LIN {X 0,Y 142.347,Z 443.787,A -85,B 0,C 180,E1 -25610.985,E2 -25610.985} C_VEL
LIN {X 0,Y 135.867,Z 450.599,A -85,B 0,C 180,E1 -25615.317,E2 -25615.317} C_VEL
LIN {X 0,Y 131.216,Z 455.128,A -85,B 0,C 180,E1 -25619.411,E2 -25619.411} C_VEL
LIN {X 0,Y 127.135,Z 458.6,A -85,B 0,C 180,E1 -25623.749,E2 -25623.749} C_VEL
LIN {X 0,Y 122.957,Z 461.7,A -85,B 0,C 180,E1 -25629.939,E2 -25629.939} C_VEL
LIN {X 0,Y 120.458,Z 463.257,A -85,B 0,C 180,E1 -25636.499,E2 -25636.499} C_VEL
LIN {X 0,Y 119.459,Z 463.204,A -85,B 0,C 180,E1 -25643.237,E2 -25643.237} C_VEL
LIN {X 0,Y 119.528,Z 462.151,A -85,B 0,C 180,E1 -25648.311,E2 -25648.311} C_VEL
LIN {X 0,Y 119.517,Z 460.979,A -85,B 0,C 180,E1 -25651.51,E2 -25651.51} C_VEL
LIN {X 0,Y 119.554,Z 458.203,A -85,B 0,C 180,E1 -25656.745,E2 -25656.745} C_VEL
LIN {X 0,Y 120.052,Z 454.435,A -85,B 0,C 180,E1 -25661.816,E2 -25661.816} C_VEL
LIN {X 0,Y 121.344,Z 449.309,A -85,B 0,C 180,E1 -25667.013,E2 -25667.013} C_VEL
LIN {X 0,Y 123.514,Z 443.317,A -85,B 0,C 180,E1 -25671.698,E2 -25671.698} C_VEL
LIN {X 0,Y 126.362,Z 435.566,A -85,B 0,C 180,E1 -25676.41,E2 -25676.41} C_VEL
LIN {X 0,Y 127.73,Z 431.92,A -85,B 0,C 180,E1 -25678.233,E2 -25678.233} C_VEL
LIN {X 0,Y 128.781,Z 427.935,A -85,B 0,C 180,E1 -25680.111,E2 -25680.111} C_VEL
LIN {X 0,Y 128.861,Z 421.063,A -85,B 0,C 180,E1 -25683.301,E2 -25683.301} C_VEL
LIN {X 0,Y 128.961,Z 413.731,A -85,B 0,C 180,E1 -25686.286,E2 -25686.286} C_VEL
LIN {X 0,Y 129.981,Z 408.956,A -85,B 0,C 180,E1 -25687.771,E2 -25687.771} C_VEL
LIN {X 0,Y 133.424,Z 398.451,A -85,B 0,C 180,E1 -25690.173,E2 -25690.173} C_VEL
LIN {X 0,Y 136.671,Z 386.681,A -85,B 0,C 180,E1 -25692.187,E2 -25692.187} C_VEL
LIN {X 0,Y 139.335,Z 373.81,A -85,B 0,C 180,E1 -25693.773,E2 -25693.773} C_VEL
LIN {X 0,Y 141.317,Z 360.485,A -85,B 0,C 180,E1 -25694.819,E2 -25694.819} C_VEL
LIN {X 0,Y 143.543,Z 329.086,A -85,B 0,C 180,E1 -25696.247,E2 -25696.247} C_VEL
LIN {X 0,Y 143.992,Z 319.506,A -85,B 0,C 180,E1 -25696.718,E2 -25696.718} C_VEL
LIN {X 0,Y 143.262,Z 306.343,A -85,B 0,C 180,E1 -25697.853,E2 -25697.853} C_VEL
LIN {X 0,Y 138.673,Z 293.214,A -85,B 0,C 180,E1 -25700.561,E2 -25700.561} C_VEL
LIN {X 0,Y 133.405,Z 281.529,A -85,B 0,C 180,E1 -25703.8,E2 -25703.8} C_VEL
LIN {X 0,Y 128.28,Z 273.681,A -85,B 0,C 180,E1 -25707.131,E2 -25707.131} C_VEL
LIN {X 0,Y 125.597,Z 269.89,A -85,B 0,C 180,E1 -25709.063,E2 -25709.063} C_VEL
LIN {X 0,Y 123.046,Z 266.259,A -85,B 0,C 180,E1 -25711.072,E2 -25711.072} C_VEL
LIN {X 0,Y 119.947,Z 262.642,A -85,B 0,C 180,E1 -25713.698,E2 -25713.698} C_VEL
LIN {X 0,Y 119.012,Z 260.746,A -85,B 0,C 180,E1 -25714.651,E2 -25714.651} C_VEL
LIN {X 0,Y 116.625,Z 258.914,A -85,B 0,C 180,E1 -25716.905,E2 -25716.905} C_VEL
LIN {X 0,Y 115.229,Z 256.404,A -85,B 0,C 180,E1 -25718.534,E2 -25718.534} C_VEL
LIN {X 0,Y 114.966,Z 255.164,A -85,B 0,C 180,E1 -25719.07,E2 -25719.07} C_VEL
LIN {X 0,Y 115.102,Z 255.137,A -85,B 0,C 180,E1 -25725.864,E2 -25725.864} C_VEL
LIN {X 0,Y 115.285,Z 255.125,A -85,B 0,C 180,E1 -25729.462,E2 -25729.462} C_VEL
LIN {X 0,Y 115.488,Z 255.097,A -85,B 0,C 180,E1 -25736.511,E2 -25736.511} C_VEL
LIN {X 0,Y 115.95,Z 254.997,A -85,B 0,C 180,E1 -25740,E2 -25740} C_VEL
LIN {X 0,Y 115.327,Z 255.113,A -85,B 0,C 180,E1 -25747.001,E2 -25747.001} C_VEL
LIN {X 0,Y 115.178,Z 255.094,A -85,B 0,C 180,E1 -25752.556,E2 -25752.556} C_VEL
LIN {X 0,Y 114.938,Z 255.142,A -85,B 0,C 180,E1 -25757.802,E2 -25757.802} C_VEL
LIN {X 0,Y 114.891,Z 255.162,A -85,B 0,C 180,E1 -25763.457,E2 -25763.457} C_VEL
LIN {X 0,Y 114.843,Z 255.178,A -85,B 0,C 180,E1 -25771.068,E2 -25771.068} C_VEL
LIN {X 0,Y 114.795,Z 255.21,A -85,B 0,C 180,E1 -25772.593,E2 -25772.593} C_VEL
LIN {X 0,Y 115.589,Z 257.654,A -85,B 0,C 180,E1 -25773.699,E2 -25773.699} C_VEL
LIN {X 0,Y 117.753,Z 260.059,A -85,B 0,C 180,E1 -25775.949,E2 -25775.949} C_VEL
LIN {X 0,Y 119.112,Z 260.981,A -85,B 0,C 180,E1 -25777.182,E2 -25777.182} C_VEL
LIN {X 0,Y 121.041,Z 264.197,A -85,B 0,C 180,E1 -25779.023,E2 -25779.023} C_VEL
LIN {X 0,Y 123.115,Z 266.362,A -85,B 0,C 180,E1 -25780.713,E2 -25780.713} C_VEL
LIN {X 0,Y 125.486,Z 269.811,A -85,B 0,C 180,E1 -25782.589,E2 -25782.589} C_VEL
LIN {X 0,Y 126.743,Z 271.497,A -85,B 0,C 180,E1 -25783.51,E2 -25783.51} C_VEL
LIN {X 0,Y 131.911,Z 279.095,A -85,B 0,C 180,E1 -25786.994,E2 -25786.994} C_VEL
LIN {X 0,Y 137.593,Z 288.613,A -85,B 0,C 180,E1 -25790.375,E2 -25790.375} C_VEL
LIN {X 0,Y 142.188,Z 297.608,A -85,B 0,C 180,E1 -25792.876,E2 -25792.876} C_VEL
LIN {X 0,Y 144.941,Z 303.696,A -85,B 0,C 180,E1 -25794.304,E2 -25794.304} C_VEL
LIN {X 0,Y 141.754,Z 350.025,A -85,B 0,C 180,E1 -25796.354,E2 -25796.354} C_VEL
LIN {X 0,Y 139.926,Z 363.432,A -85,B 0,C 180,E1 -25797.438,E2 -25797.438} C_VEL
LIN {X 0,Y 137.503,Z 376.255,A -85,B 0,C 180,E1 -25799.058,E2 -25799.058} C_VEL
LIN {X 0,Y 134.688,Z 387.934,A -85,B 0,C 180,E1 -25801.15,E2 -25801.15} C_VEL
LIN {X 0,Y 131.103,Z 399.265,A -85,B 0,C 180,E1 -25803.761,E2 -25803.761} C_VEL
LIN {X 0,Y 127.423,Z 409.472,A -85,B 0,C 180,E1 -25806.869,E2 -25806.869} C_VEL
LIN {X 0,Y 124.118,Z 417.825,A -85,B 0,C 180,E1 -25810.147,E2 -25810.147} C_VEL
LIN {X 0,Y 120.414,Z 426.872,A -85,B 0,C 180,E1 -25814.781,E2 -25814.781} C_VEL
LIN {X 0,Y 117.233,Z 434.194,A -85,B 0,C 180,E1 -25819.647,E2 -25819.647} C_VEL
LIN {X 0,Y 115.036,Z 440.041,A -85,B 0,C 180,E1 -25824.749,E2 -25824.749} C_VEL
LIN {X 0,Y 113.521,Z 444.662,A -85,B 0,C 180,E1 -25830.007,E2 -25830.007} C_VEL
LIN {X 0,Y 112.764,Z 447.542,A -85,B 0,C 180,E1 -25834.285,E2 -25834.285} C_VEL
LIN {X 0,Y 112.166,Z 450.75,A -85,B 0,C 180,E1 -25840.84,E2 -25840.84} C_VEL
LIN {X 0,Y 112.34,Z 451.922,A -85,B 0,C 180,E1 -25844.497,E2 -25844.497} C_VEL
LIN {X 0,Y 112.924,Z 452.662,A -85,B 0,C 180,E1 -25848.136,E2 -25848.136} C_VEL
LIN {X 0,Y 113.99,Z 453.051,A -85,B 0,C 180,E1 -25852.357,E2 -25852.357} C_VEL
LIN {X 0,Y 116.639,Z 452.5,A -85,B 0,C 180,E1 -25858.823,E2 -25858.823} C_VEL
LIN {X 0,Y 118.635,Z 451.603,A -85,B 0,C 180,E1 -25862.223,E2 -25862.223} C_VEL
LIN {X 0,Y 121.126,Z 450.227,A -85,B 0,C 180,E1 -25865.676,E2 -25865.676} C_VEL
LIN {X 0,Y 125.185,Z 447.493,A -85,B 0,C 180,E1 -25870.216,E2 -25870.216} C_VEL
LIN {X 0,Y 130.145,Z 443.612,A -85,B 0,C 180,E1 -25874.592,E2 -25874.592} C_VEL
LIN {X 0,Y 136.739,Z 437.557,A -85,B 0,C 180,E1 -25879.3,E2 -25879.3} C_VEL
LIN {X 0,Y 143.074,Z 430.847,A -85,B 0,C 180,E1 -25882.962,E2 -25882.962} C_VEL
LIN {X 0,Y 148.716,Z 423.972,A -85,B 0,C 180,E1 -25885.791,E2 -25885.791} C_VEL
LIN {X 0,Y 154.702,Z 415.627,A -85,B 0,C 180,E1 -25888.408,E2 -25888.408} C_VEL
LIN {X 0,Y 160.312,Z 406.479,A -85,B 0,C 180,E1 -25890.611,E2 -25890.611} C_VEL
LIN {X 0,Y 166.148,Z 395.072,A -85,B 0,C 180,E1 -25892.658,E2 -25892.658} C_VEL
LIN {X 0,Y 170.694,Z 383.759,A -85,B 0,C 180,E1 -25894.244,E2 -25894.244} C_VEL
LIN {X 0,Y 174.645,Z 371.716,A -85,B 0,C 180,E1 -25895.405,E2 -25895.405} C_VEL
LIN {X 0,Y 177.667,Z 358.526,A -85,B 0,C 180,E1 -25896.32,E2 -25896.32} C_VEL
LIN {X 0,Y 179.589,Z 345.087,A -85,B 0,C 180,E1 -25896.904,E2 -25896.904} C_VEL
LIN {X 0,Y 180.483,Z 334.894,A -85,B 0,C 180,E1 -25897.234,E2 -25897.234} C_VEL
LIN {X 0,Y 176.224,Z 326.44,A -85,B 0,C 180,E1 -25900.715,E2 -25900.715} C_VEL
LIN {X 0,Y 172.654,Z 319.94,A -85,B 0,C 180,E1 -25904.128,E2 -25904.128} C_VEL
LIN {X 0,Y 170.098,Z 315.805,A -85,B 0,C 180,E1 -25906.979,E2 -25906.979} C_VEL
LIN {X 0,Y 168.062,Z 312.363,A -85,B 0,C 180,E1 -25909.724,E2 -25909.724} C_VEL
LIN {X 0,Y 165.797,Z 308.448,A -85,B 0,C 180,E1 -25913.611,E2 -25913.611} C_VEL
LIN {X 0,Y 163.767,Z 305.133,A -85,B 0,C 180,E1 -25918.942,E2 -25918.942} C_VEL
LIN {X 0,Y 163.452,Z 303.929,A -85,B 0,C 180,E1 -25920.616,E2 -25920.616} C_VEL
LIN {X 0,Y 163.384,Z 304.122,A -85,B 0,C 180,E1 -25929.602,E2 -25929.602} C_VEL
LIN {X 0,Y 164.811,Z 307.662,A -85,B 0,C 180,E1 -25934.824,E2 -25934.824} C_VEL
LIN {X 0,Y 166.15,Z 309.281,A -85,B 0,C 180,E1 -25937.54,E2 -25937.54} C_VEL
LIN {X 0,Y 168.65,Z 314.118,A -85,B 0,C 180,E1 -25941.652,E2 -25941.652} C_VEL
LIN {X 0,Y 171.028,Z 319.175,A -85,B 0,C 180,E1 -25944.763,E2 -25944.763} C_VEL
LIN {X 0,Y 173.756,Z 325.357,A -85,B 0,C 180,E1 -25947.77,E2 -25947.77} C_VEL
LIN {X 0,Y 176.936,Z 333.399,A -85,B 0,C 180,E1 -25950.84,E2 -25950.84} C_VEL
LIN {X 0,Y 179.897,Z 341.767,A -85,B 0,C 180,E1 -25953.41,E2 -25953.41} C_VEL
LIN {X 0,Y 178.104,Z 359.854,A -85,B 0,C 180,E1 -25954.039,E2 -25954.039} C_VEL
LIN {X 0,Y 175.568,Z 372.981,A -85,B 0,C 180,E1 -25954.697,E2 -25954.697} C_VEL
LIN {X 0,Y 172.279,Z 384.753,A -85,B 0,C 180,E1 -25955.577,E2 -25955.577} C_VEL
LIN {X 0,Y 167.768,Z 396.618,A -85,B 0,C 180,E1 -25956.758,E2 -25956.758} C_VEL
LIN {X 0,Y 162.377,Z 408.014,A -85,B 0,C 180,E1 -25958.327,E2 -25958.327} C_VEL
LIN {X 0,Y 157.198,Z 417.236,A -85,B 0,C 180,E1 -25960.037,E2 -25960.037} C_VEL
LIN {X 0,Y 151.494,Z 425.849,A -85,B 0,C 180,E1 -25962.075,E2 -25962.075} C_VEL
LIN {X 0,Y 145.657,Z 433.793,A -85,B 0,C 180,E1 -25964.625,E2 -25964.625} C_VEL
LIN {X 0,Y 139.037,Z 441.612,A -85,B 0,C 180,E1 -25967.95,E2 -25967.95} C_VEL
LIN {X 0,Y 133.839,Z 446.946,A -85,B 0,C 180,E1 -25970.938,E2 -25970.938} C_VEL
LIN {X 0,Y 128.183,Z 452.339,A -85,B 0,C 180,E1 -25975.04,E2 -25975.04} C_VEL
LIN {X 0,Y 123.637,Z 456.276,A -85,B 0,C 180,E1 -25979.226,E2 -25979.226} C_VEL
LIN {X 0,Y 120.79,Z 458.43,A -85,B 0,C 180,E1 -25982.255,E2 -25982.255} C_VEL
LIN {X 0,Y 116.295,Z 461.47,A -85,B 0,C 180,E1 -25988.735,E2 -25988.735} C_VEL
LIN {X 0,Y 114.689,Z 462.412,A -85,B 0,C 180,E1 -25992.153,E2 -25992.153} C_VEL
LIN {X 0,Y 113.553,Z 462.948,A -85,B 0,C 180,E1 -25995.661,E2 -25995.661} C_VEL
LIN {X 0,Y 112.409,Z 462.834,A -85,B 0,C 180,E1 -26002.811,E2 -26002.811} C_VEL
LIN {X 0,Y 112.481,Z 461.606,A -85,B 0,C 180,E1 -26008.608,E2 -26008.608} C_VEL
LIN {X 0,Y 112.404,Z 459.646,A -85,B 0,C 180,E1 -26013.578,E2 -26013.578} C_VEL
LIN {X 0,Y 112.594,Z 456.537,A -85,B 0,C 180,E1 -26018.97,E2 -26018.97} C_VEL
LIN {X 0,Y 113.431,Z 452.33,A -85,B 0,C 180,E1 -26024.341,E2 -26024.341} C_VEL
LIN {X 0,Y 115.588,Z 445.905,A -85,B 0,C 180,E1 -26030.454,E2 -26030.454} C_VEL
LIN {X 0,Y 118.348,Z 438.885,A -85,B 0,C 180,E1 -26035.492,E2 -26035.492} C_VEL
LIN {X 0,Y 121.412,Z 431.224,A -85,B 0,C 180,E1 -26039.74,E2 -26039.74} C_VEL
LIN {X 0,Y 124.822,Z 422.996,A -85,B 0,C 180,E1 -26043.285,E2 -26043.285} C_VEL
LIN {X 0,Y 128.267,Z 413.406,A -85,B 0,C 180,E1 -26046.563,E2 -26046.563} C_VEL
LIN {X 0,Y 129.981,Z 408.956,A -85,B 0,C 180,E1 -26047.771,E2 -26047.771} C_VEL
LIN {X 0,Y 131.01,Z 404.106,A -85,B 0,C 180,E1 -26049.141,E2 -26049.141} C_VEL
LIN {X 0,Y 131.222,Z 395.906,A -85,B 0,C 180,E1 -26051.563,E2 -26051.563} C_VEL
LIN {X 0,Y 131.355,Z 387.318,A -85,B 0,C 180,E1 -26053.743,E2 -26053.743} C_VEL
LIN {X 0,Y 132.174,Z 381.808,A -85,B 0,C 180,E1 -26054.695,E2 -26054.695} C_VEL
LIN {X 0,Y 134.706,Z 368.977,A -85,B 0,C 180,E1 -26056.093,E2 -26056.093} C_VEL
LIN {X 0,Y 136.259,Z 356.658,A -85,B 0,C 180,E1 -26056.957,E2 -26056.957} C_VEL
LIN {X 0,Y 138.731,Z 320.833,A -85,B 0,C 180,E1 -26058.568,E2 -26058.568} C_VEL
LIN {X 0,Y 138.158,Z 308.787,A -85,B 0,C 180,E1 -26059.649,E2 -26059.649} C_VEL
LIN {X 0,Y 133.929,Z 296.482,A -85,B 0,C 180,E1 -26062.379,E2 -26062.379} C_VEL
LIN {X 0,Y 129.496,Z 286.224,A -85,B 0,C 180,E1 -26065.378,E2 -26065.378} C_VEL
LIN {X 0,Y 124.317,Z 278.18,A -85,B 0,C 180,E1 -26069.063,E2 -26069.063} C_VEL
LIN {X 0,Y 122.2,Z 275.163,A -85,B 0,C 180,E1 -26070.735,E2 -26070.735} C_VEL
LIN {X 0,Y 119.662,Z 271.528,A -85,B 0,C 180,E1 -26072.924,E2 -26072.924} C_VEL
LIN {X 0,Y 117.151,Z 268.278,A -85,B 0,C 180,E1 -26075.288,E2 -26075.288} C_VEL
LIN {X 0,Y 116.364,Z 266.998,A -85,B 0,C 180,E1 -26076.119,E2 -26076.119} C_VEL
LIN {X 0,Y 113.899,Z 264.457,A -85,B 0,C 180,E1 -26078.746,E2 -26078.746} C_VEL
LIN {X 0,Y 112.644,Z 261.908,A -85,B 0,C 180,E1 -26080.406,E2 -26080.406} C_VEL
LIN {X 0,Y 109.73,Z 259.907,A -85,B 0,C 180,E1 -26084.205,E2 -26084.205} C_VEL
LIN {X 0,Y 108.446,Z 257.52,A -85,B 0,C 180,E1 -26086.465,E2 -26086.465} C_VEL
LIN {X 0,Y 108.162,Z 256,A -85,B 0,C 180,E1 -26087.355,E2 -26087.355} C_VEL
LIN {X 0,Y 108.271,Z 255.985,A -85,B 0,C 180,E1 -26092.541,E2 -26092.541} C_VEL
LIN {X 0,Y 108.876,Z 255.876,A -85,B 0,C 180,E1 -26100,E2 -26100} C_VEL
LIN {X 0,Y 108.266,Z 255.994,A -85,B 0,C 180,E1 -26107.46,E2 -26107.46} C_VEL
LIN {X 0,Y 108.113,Z 255.97,A -85,B 0,C 180,E1 -26112.871,E2 -26112.871} C_VEL
LIN {X 0,Y 107.837,Z 256.042,A -85,B 0,C 180,E1 -26119.018,E2 -26119.018} C_VEL
LIN {X 0,Y 107.84,Z 256.152,A -85,B 0,C 180,E1 -26124.036,E2 -26124.036} C_VEL
LIN {X 0,Y 108.529,Z 258.484,A -85,B 0,C 180,E1 -26125.582,E2 -26125.582} C_VEL
LIN {X 0,Y 110.392,Z 260.745,A -85,B 0,C 180,E1 -26128.522,E2 -26128.522} C_VEL
LIN {X 0,Y 112.556,Z 262.103,A -85,B 0,C 180,E1 -26131.249,E2 -26131.249} C_VEL
LIN {X 0,Y 114.14,Z 264.967,A -85,B 0,C 180,E1 -26133.283,E2 -26133.283} C_VEL
LIN {X 0,Y 116.728,Z 267.477,A -85,B 0,C 180,E1 -26135.98,E2 -26135.98} C_VEL
LIN {X 0,Y 118.956,Z 270.795,A -85,B 0,C 180,E1 -26138.183,E2 -26138.183} C_VEL
LIN {X 0,Y 120.503,Z 272.706,A -85,B 0,C 180,E1 -26139.549,E2 -26139.549} C_VEL
LIN {X 0,Y 123.972,Z 277.674,A -85,B 0,C 180,E1 -26142.397,E2 -26142.397} C_VEL
LIN {X 0,Y 129.166,Z 285.657,A -85,B 0,C 180,E1 -26146.127,E2 -26146.127} C_VEL
LIN {X 0,Y 134.683,Z 295.4,A -85,B 0,C 180,E1 -26149.608,E2 -26149.608} C_VEL
LIN {X 0,Y 139.641,Z 306.063,A -85,B 0,C 180,E1 -26152.474,E2 -26152.474} C_VEL
LIN {X 0,Y 136.453,Z 349.707,A -85,B 0,C 180,E1 -26154.409,E2 -26154.409} C_VEL
LIN {X 0,Y 134.551,Z 363.306,A -85,B 0,C 180,E1 -26155.511,E2 -26155.511} C_VEL
LIN {X 0,Y 131.991,Z 376.282,A -85,B 0,C 180,E1 -26157.16,E2 -26157.16} C_VEL
LIN {X 0,Y 129.021,Z 388.023,A -85,B 0,C 180,E1 -26159.302,E2 -26159.302} C_VEL
LIN {X 0,Y 125.248,Z 399.397,A -85,B 0,C 180,E1 -26161.979,E2 -26161.979} C_VEL
LIN {X 0,Y 121.345,Z 409.647,A -85,B 0,C 180,E1 -26165.181,E2 -26165.181} C_VEL
LIN {X 0,Y 117.481,Z 418.844,A -85,B 0,C 180,E1 -26168.974,E2 -26168.974} C_VEL
LIN {X 0,Y 113.579,Z 427.776,A -85,B 0,C 180,E1 -26173.841,E2 -26173.841} C_VEL
LIN {X 0,Y 110.261,Z 434.994,A -85,B 0,C 180,E1 -26178.984,E2 -26178.984} C_VEL
LIN {X 0,Y 107.961,Z 440.736,A -85,B 0,C 180,E1 -26184.404,E2 -26184.404} C_VEL
LIN {X 0,Y 106.406,Z 445.269,A -85,B 0,C 180,E1 -26190.007,E2 -26190.007} C_VEL
LIN {X 0,Y 105.692,Z 447.832,A -85,B 0,C 180,E1 -26194.1,E2 -26194.1} C_VEL
LIN {X 0,Y 105.097,Z 451.232,A -85,B 0,C 180,E1 -26201.579,E2 -26201.579} C_VEL
LIN {X 0,Y 105.343,Z 452.342,A -85,B 0,C 180,E1 -26205.484,E2 -26205.484} C_VEL
LIN {X 0,Y 106.033,Z 453.049,A -85,B 0,C 180,E1 -26209.36,E2 -26209.36} C_VEL
LIN {X 0,Y 107.122,Z 453.374,A -85,B 0,C 180,E1 -26213.29,E2 -26213.29} C_VEL
LIN {X 0,Y 108.473,Z 453.282,A -85,B 0,C 180,E1 -26216.976,E2 -26216.976} C_VEL
LIN {X 0,Y 112.524,Z 451.816,A -85,B 0,C 180,E1 -26224.207,E2 -26224.207} C_VEL
LIN {X 0,Y 115.129,Z 450.478,A -85,B 0,C 180,E1 -26227.626,E2 -26227.626} C_VEL
LIN {X 0,Y 119.687,Z 447.6,A -85,B 0,C 180,E1 -26232.479,E2 -26232.479} C_VEL
LIN {X 0,Y 125.039,Z 443.643,A -85,B 0,C 180,E1 -26236.947,E2 -26236.947} C_VEL
LIN {X 0,Y 132.088,Z 437.464,A -85,B 0,C 180,E1 -26241.705,E2 -26241.705} C_VEL
LIN {X 0,Y 138.762,Z 430.698,A -85,B 0,C 180,E1 -26245.35,E2 -26245.35} C_VEL
LIN {X 0,Y 144.741,Z 423.673,A -85,B 0,C 180,E1 -26248.182,E2 -26248.182} C_VEL
LIN {X 0,Y 151.02,Z 415.206,A -85,B 0,C 180,E1 -26250.759,E2 -26250.759} C_VEL
LIN {X 0,Y 156.882,Z 405.887,A -85,B 0,C 180,E1 -26252.918,E2 -26252.918} C_VEL
LIN {X 0,Y 162.906,Z 394.188,A -85,B 0,C 180,E1 -26254.953,E2 -26254.953} C_VEL
LIN {X 0,Y 167.659,Z 382.594,A -85,B 0,C 180,E1 -26256.485,E2 -26256.485} C_VEL
LIN {X 0,Y 171.744,Z 369.884,A -85,B 0,C 180,E1 -26257.618,E2 -26257.618} C_VEL
LIN {X 0,Y 174.691,Z 356.619,A -85,B 0,C 180,E1 -26258.471,E2 -26258.471} C_VEL
LIN {X 0,Y 176.52,Z 342.976,A -85,B 0,C 180,E1 -26258.987,E2 -26258.987} C_VEL
LIN {X 0,Y 176.921,Z 338.494,A -85,B 0,C 180,E1 -26259.128,E2 -26259.128} C_VEL
LIN {X 0,Y 173.125,Z 330.723,A -85,B 0,C 180,E1 -26262.579,E2 -26262.579} C_VEL
LIN {X 0,Y 169.977,Z 324.839,A -85,B 0,C 180,E1 -26265.941,E2 -26265.941} C_VEL
LIN {X 0,Y 166.883,Z 319.326,A -85,B 0,C 180,E1 -26270.072,E2 -26270.072} C_VEL
LIN {X 0,Y 164.576,Z 315.251,A -85,B 0,C 180,E1 -26274.234,E2 -26274.234} C_VEL
LIN {X 0,Y 162.653,Z 311.604,A -85,B 0,C 180,E1 -26280,E2 -26280} C_VEL
LIN {X 0,Y 162.451,Z 310.898,A -85,B 0,C 180,E1 -26281.239,E2 -26281.239} C_VEL
LIN {X 0,Y 162.453,Z 311.16,A -85,B 0,C 180,E1 -26289.336,E2 -26289.336} C_VEL
LIN {X 0,Y 163.82,Z 314.679,A -85,B 0,C 180,E1 -26294.598,E2 -26294.598} C_VEL
LIN {X 0,Y 164.888,Z 316.052,A -85,B 0,C 180,E1 -26296.896,E2 -26296.896} C_VEL
LIN {X 0,Y 167.035,Z 320.457,A -85,B 0,C 180,E1 -26300.713,E2 -26300.713} C_VEL
LIN {X 0,Y 169.118,Z 325.207,A -85,B 0,C 180,E1 -26303.688,E2 -26303.688} C_VEL
LIN {X 0,Y 171.581,Z 331.255,A -85,B 0,C 180,E1 -26306.65,E2 -26306.65} C_VEL
LIN {X 0,Y 174.74,Z 339.727,A -85,B 0,C 180,E1 -26309.932,E2 -26309.932} C_VEL
LIN {X 0,Y 176.339,Z 344.663,A -85,B 0,C 180,E1 -26311.467,E2 -26311.467} C_VEL
LIN {X 0,Y 174.682,Z 360.164,A -85,B 0,C 180,E1 -26312.021,E2 -26312.021} C_VEL
LIN {X 0,Y 172.126,Z 372.876,A -85,B 0,C 180,E1 -26312.652,E2 -26312.652} C_VEL
LIN {X 0,Y 168.625,Z 384.899,A -85,B 0,C 180,E1 -26313.534,E2 -26313.534} C_VEL
LIN {X 0,Y 163.648,Z 397.438,A -85,B 0,C 180,E1 -26314.781,E2 -26314.781} C_VEL
LIN {X 0,Y 158.096,Z 408.626,A -85,B 0,C 180,E1 -26316.319,E2 -26316.319} C_VEL
LIN {X 0,Y 152.067,Z 418.717,A -85,B 0,C 180,E1 -26318.216,E2 -26318.216} C_VEL
LIN {X 0,Y 145.655,Z 427.832,A -85,B 0,C 180,E1 -26320.538,E2 -26320.538} C_VEL
LIN {X 0,Y 138.406,Z 436.735,A -85,B 0,C 180,E1 -26323.647,E2 -26323.647} C_VEL
LIN {X 0,Y 131.612,Z 443.928,A -85,B 0,C 180,E1 -26327.088,E2 -26327.088} C_VEL
LIN {X 0,Y 126.364,Z 448.803,A -85,B 0,C 180,E1 -26330.235,E2 -26330.235} C_VEL
LIN {X 0,Y 120.518,Z 453.852,A -85,B 0,C 180,E1 -26334.726,E2 -26334.726} C_VEL
LIN {X 0,Y 116.038,Z 457.251,A -85,B 0,C 180,E1 -26339.011,E2 -26339.011} C_VEL
LIN {X 0,Y 111.953,Z 459.947,A -85,B 0,C 180,E1 -26343.927,E2 -26343.927} C_VEL
LIN {X 0,Y 107.912,Z 462.146,A -85,B 0,C 180,E1 -26350.991,E2 -26350.991} C_VEL
LIN {X 0,Y 105.775,Z 462.736,A -85,B 0,C 180,E1 -26358.496,E2 -26358.496} C_VEL
LIN {X 0,Y 105.315,Z 461.812,A -85,B 0,C 180,E1 -26366.167,E2 -26366.167} C_VEL
LIN {X 0,Y 105.423,Z 460.559,A -85,B 0,C 180,E1 -26370.422,E2 -26370.422} C_VEL
LIN {X 0,Y 105.321,Z 459.162,A -85,B 0,C 180,E1 -26373.819,E2 -26373.819} C_VEL
LIN {X 0,Y 105.552,Z 455.988,A -85,B 0,C 180,E1 -26379.574,E2 -26379.574} C_VEL
LIN {X 0,Y 106.513,Z 451.714,A -85,B 0,C 180,E1 -26385.295,E2 -26385.295} C_VEL
LIN {X 0,Y 108.473,Z 446.237,A -85,B 0,C 180,E1 -26390.866,E2 -26390.866} C_VEL
LIN {X 0,Y 111.341,Z 439.369,A -85,B 0,C 180,E1 -26396.212,E2 -26396.212} C_VEL
LIN {X 0,Y 114.933,Z 431.092,A -85,B 0,C 180,E1 -26401.121,E2 -26401.121} C_VEL
LIN {X 0,Y 118.894,Z 421.971,A -85,B 0,C 180,E1 -26405.182,E2 -26405.182} C_VEL
LIN {X 0,Y 122.62,Z 412.248,A -85,B 0,C 180,E1 -26408.545,E2 -26408.545} C_VEL
LIN {X 0,Y 126.607,Z 401.696,A -85,B 0,C 180,E1 -26411.225,E2 -26411.225} C_VEL
LIN {X 0,Y 129.641,Z 391.817,A -85,B 0,C 180,E1 -26413.176,E2 -26413.176} C_VEL
LIN {X 0,Y 132.174,Z 381.808,A -85,B 0,C 180,E1 -26414.695,E2 -26414.695} C_VEL
LIN {X 0,Y 132.862,Z 376.285,A -85,B 0,C 180,E1 -26415.562,E2 -26415.562} C_VEL
LIN {X 0,Y 132.287,Z 367.186,A -85,B 0,C 180,E1 -26417.265,E2 -26417.265} C_VEL
LIN {X 0,Y 131.384,Z 357.905,A -85,B 0,C 180,E1 -26418.753,E2 -26418.753} C_VEL
LIN {X 0,Y 131.43,Z 352.096,A -85,B 0,C 180,E1 -26419.242,E2 -26419.242} C_VEL
LIN {X 0,Y 133.601,Z 321.52,A -85,B 0,C 180,E1 -26420.615,E2 -26420.615} C_VEL
LIN {X 0,Y 133.201,Z 311.294,A -85,B 0,C 180,E1 -26421.566,E2 -26421.566} C_VEL
LIN {X 0,Y 129.315,Z 299.601,A -85,B 0,C 180,E1 -26424.346,E2 -26424.346} C_VEL
LIN {X 0,Y 125.65,Z 290.946,A -85,B 0,C 180,E1 -26427.074,E2 -26427.074} C_VEL
LIN {X 0,Y 121.157,Z 283.62,A -85,B 0,C 180,E1 -26430.577,E2 -26430.577} C_VEL
LIN {X 0,Y 117.013,Z 277.535,A -85,B 0,C 180,E1 -26434.301,E2 -26434.301} C_VEL
LIN {X 0,Y 114.363,Z 273.751,A -85,B 0,C 180,E1 -26437.055,E2 -26437.055} C_VEL
LIN {X 0,Y 111.286,Z 269.933,A -85,B 0,C 180,E1 -26440.697,E2 -26440.697} C_VEL
LIN {X 0,Y 110.421,Z 268.388,A -85,B 0,C 180,E1 -26441.924,E2 -26441.924} C_VEL
LIN {X 0,Y 107.789,Z 266.13,A -85,B 0,C 180,E1 -26445.753,E2 -26445.753} C_VEL
LIN {X 0,Y 106.447,Z 263.156,A -85,B 0,C 180,E1 -26448.501,E2 -26448.501} C_VEL
LIN {X 0,Y 106.191,Z 262.809,A -85,B 0,C 180,E1 -26449.032,E2 -26449.032} C_VEL
LIN {X 0,Y 103.149,Z 260.666,A -85,B 0,C 180,E1 -26457.071,E2 -26457.071} C_VEL
LIN {X 0,Y 102.648,Z 259.347,A -85,B 0,C 180,E1 -26460,E2 -26460} C_VEL
LIN {X 0,Y 102.206,Z 259.828,A -85,B 0,C 180,E1 -26468.901,E2 -26468.901} C_VEL
LIN {X 0,Y 103.263,Z 261.362,A -85,B 0,C 180,E1 -26475.356,E2 -26475.356} C_VEL
LIN {X 0,Y 106.181,Z 263.133,A -85,B 0,C 180,E1 -26482.755,E2 -26482.755} C_VEL
LIN {X 0,Y 107.454,Z 266.002,A -85,B 0,C 180,E1 -26485.458,E2 -26485.458} C_VEL
LIN {X 0,Y 109.916,Z 268.218,A -85,B 0,C 180,E1 -26489.179,E2 -26489.179} C_VEL
LIN {X 0,Y 110.563,Z 268.78,A -85,B 0,C 180,E1 -26490.039,E2 -26490.039} C_VEL
LIN {X 0,Y 112.644,Z 272.024,A -85,B 0,C 180,E1 -26492.768,E2 -26492.768} C_VEL
LIN {X 0,Y 114.413,Z 273.877,A -85,B 0,C 180,E1 -26494.729,E2 -26494.729} C_VEL
LIN {X 0,Y 117.187,Z 277.71,A -85,B 0,C 180,E1 -26497.582,E2 -26497.582} C_VEL
LIN {X 0,Y 121.175,Z 283.69,A -85,B 0,C 180,E1 -26501.167,E2 -26501.167} C_VEL
LIN {X 0,Y 126.484,Z 292.328,A -85,B 0,C 180,E1 -26505.249,E2 -26505.249} C_VEL
LIN {X 0,Y 131.407,Z 301.629,A -85,B 0,C 180,E1 -26508.576,E2 -26508.576} C_VEL
LIN {X 0,Y 134.408,Z 308.349,A -85,B 0,C 180,E1 -26510.472,E2 -26510.472} C_VEL
LIN {X 0,Y 131.239,Z 349.999,A -85,B 0,C 180,E1 -26512.357,E2 -26512.357} C_VEL
LIN {X 0,Y 129.338,Z 363.121,A -85,B 0,C 180,E1 -26513.426,E2 -26513.426} C_VEL
LIN {X 0,Y 126.64,Z 376.258,A -85,B 0,C 180,E1 -26515.1,E2 -26515.1} C_VEL
LIN {X 0,Y 123.502,Z 388.087,A -85,B 0,C 180,E1 -26517.286,E2 -26517.286} C_VEL
LIN {X 0,Y 119.526,Z 399.51,A -85,B 0,C 180,E1 -26520.025,E2 -26520.025} C_VEL
LIN {X 0,Y 115.383,Z 409.806,A -85,B 0,C 180,E1 -26523.317,E2 -26523.317} C_VEL
LIN {X 0,Y 111.684,Z 418.212,A -85,B 0,C 180,E1 -26526.85,E2 -26526.85} C_VEL
LIN {X 0,Y 107.437,Z 427.315,A -85,B 0,C 180,E1 -26531.907,E2 -26531.907} C_VEL
LIN {X 0,Y 103.793,Z 434.675,A -85,B 0,C 180,E1 -26537.296,E2 -26537.296} C_VEL
LIN {X 0,Y 101.612,Z 439.648,A -85,B 0,C 180,E1 -26542.057,E2 -26542.057} C_VEL
LIN {X 0,Y 99.682,Z 444.492,A -85,B 0,C 180,E1 -26547.988,E2 -26547.988} C_VEL
LIN {X 0,Y 98.565,Z 448.231,A -85,B 0,C 180,E1 -26554.096,E2 -26554.096} C_VEL
LIN {X 0,Y 98.063,Z 450.187,A -85,B 0,C 180,E1 -26558.248,E2 -26558.248} C_VEL
LIN {X 0,Y 98.014,Z 451.692,A -85,B 0,C 180,E1 -26562.429,E2 -26562.429} C_VEL
LIN {X 0,Y 99.199,Z 453.435,A -85,B 0,C 180,E1 -26570.753,E2 -26570.753} C_VEL
LIN {X 0,Y 100.437,Z 453.72,A -85,B 0,C 180,E1 -26574.83,E2 -26574.83} C_VEL
LIN {X 0,Y 102.007,Z 453.567,A -85,B 0,C 180,E1 -26578.84,E2 -26578.84} C_VEL
LIN {X 0,Y 106.545,Z 452.033,A -85,B 0,C 180,E1 -26586.422,E2 -26586.422} C_VEL
LIN {X 0,Y 109.424,Z 450.646,A -85,B 0,C 180,E1 -26589.966,E2 -26589.966} C_VEL
LIN {X 0,Y 114.393,Z 447.7,A -85,B 0,C 180,E1 -26594.957,E2 -26594.957} C_VEL
LIN {X 0,Y 121.681,Z 442.457,A -85,B 0,C 180,E1 -26600.555,E2 -26600.555} C_VEL
LIN {X 0,Y 128.85,Z 436.351,A -85,B 0,C 180,E1 -26604.903,E2 -26604.903} C_VEL
LIN {X 0,Y 135.587,Z 429.622,A -85,B 0,C 180,E1 -26608.306,E2 -26608.306} C_VEL
LIN {X 0,Y 142.316,Z 421.774,A -85,B 0,C 180,E1 -26611.23,E2 -26611.23} C_VEL
LIN {X 0,Y 149.602,Z 411.781,A -85,B 0,C 180,E1 -26613.956,E2 -26613.956} C_VEL
LIN {X 0,Y 155.12,Z 402.796,A -85,B 0,C 180,E1 -26615.78,E2 -26615.78} C_VEL
LIN {X 0,Y 160.637,Z 391.779,A -85,B 0,C 180,E1 -26617.552,E2 -26617.552} C_VEL
LIN {X 0,Y 165.269,Z 380.295,A -85,B 0,C 180,E1 -26618.887,E2 -26618.887} C_VEL
LIN {X 0,Y 169.246,Z 367.519,A -85,B 0,C 180,E1 -26619.93,E2 -26619.93} C_VEL
LIN {X 0,Y 171.888,Z 355.065,A -85,B 0,C 180,E1 -26620.66,E2 -26620.66} C_VEL
LIN {X 0,Y 173.481,Z 341.992,A -85,B 0,C 180,E1 -26621.166,E2 -26621.166} C_VEL
LIN {X 0,Y 170.083,Z 334.786,A -85,B 0,C 180,E1 -26624.65,E2 -26624.65} C_VEL
LIN {X 0,Y 167.319,Z 329.455,A -85,B 0,C 180,E1 -26628.03,E2 -26628.03} C_VEL
LIN {X 0,Y 165.077,Z 325.406,A -85,B 0,C 180,E1 -26631.43,E2 -26631.43} C_VEL
LIN {X 0,Y 163.287,Z 321.937,A -85,B 0,C 180,E1 -26635.062,E2 -26635.062} C_VEL
LIN {X 0,Y 161.617,Z 318.193,A -85,B 0,C 180,E1 -26640.903,E2 -26640.903} C_VEL
LIN {X 0,Y 161.371,Z 317.877,A -85,B 0,C 180,E1 -26642.496,E2 -26642.496} C_VEL
LIN {X 0,Y 161.522,Z 318.239,A -85,B 0,C 180,E1 -26649.075,E2 -26649.075} C_VEL
LIN {X 0,Y 162.742,Z 321.573,A -85,B 0,C 180,E1 -26654.138,E2 -26654.138} C_VEL
LIN {X 0,Y 163.724,Z 322.991,A -85,B 0,C 180,E1 -26656.406,E2 -26656.406} C_VEL
LIN {X 0,Y 165.566,Z 327.057,A -85,B 0,C 180,E1 -26659.932,E2 -26659.932} C_VEL
LIN {X 0,Y 167.367,Z 331.547,A -85,B 0,C 180,E1 -26662.736,E2 -26662.736} C_VEL
LIN {X 0,Y 169.581,Z 337.42,A -85,B 0,C 180,E1 -26665.63,E2 -26665.63} C_VEL
LIN {X 0,Y 172.304,Z 345.373,A -85,B 0,C 180,E1 -26668.72,E2 -26668.72} C_VEL
LIN {X 0,Y 172.984,Z 347.645,A -85,B 0,C 180,E1 -26669.449,E2 -26669.449} C_VEL
LIN {X 0,Y 171.305,Z 361.613,A -85,B 0,C 180,E1 -26669.97,E2 -26669.97} C_VEL
LIN {X 0,Y 168.498,Z 374.336,A -85,B 0,C 180,E1 -26670.621,E2 -26670.621} C_VEL
LIN {X 0,Y 164.824,Z 386.017,A -85,B 0,C 180,E1 -26671.484,E2 -26671.484} C_VEL
LIN {X 0,Y 159.726,Z 398.259,A -85,B 0,C 180,E1 -26672.7,E2 -26672.7} C_VEL
LIN {X 0,Y 154.022,Z 409.212,A -85,B 0,C 180,E1 -26674.204,E2 -26674.204} C_VEL
LIN {X 0,Y 147.799,Z 419.099,A -85,B 0,C 180,E1 -26676.062,E2 -26676.062} C_VEL
LIN {X 0,Y 141.135,Z 428.098,A -85,B 0,C 180,E1 -26678.343,E2 -26678.343} C_VEL
LIN {X 0,Y 133.611,Z 436.901,A -85,B 0,C 180,E1 -26681.446,E2 -26681.446} C_VEL
LIN {X 0,Y 126.516,Z 443.986,A -85,B 0,C 180,E1 -26684.903,E2 -26684.903} C_VEL
LIN {X 0,Y 120.982,Z 448.805,A -85,B 0,C 180,E1 -26688.08,E2 -26688.08} C_VEL
LIN {X 0,Y 114.29,Z 454.131,A -85,B 0,C 180,E1 -26693.073,E2 -26693.073} C_VEL
LIN {X 0,Y 108.401,Z 458.094,A -85,B 0,C 180,E1 -26698.752,E2 -26698.752} C_VEL
LIN {X 0,Y 103.168,Z 461.015,A -85,B 0,C 180,E1 -26705.869,E2 -26705.869} C_VEL
LIN {X 0,Y 101.19,Z 461.866,A -85,B 0,C 180,E1 -26709.674,E2 -26709.674} C_VEL
LIN {X 0,Y 98.821,Z 462.394,A -85,B 0,C 180,E1 -26717.674,E2 -26717.674} C_VEL
LIN {X 0,Y 98.224,Z 461.404,A -85,B 0,C 180,E1 -26725.89,E2 -26725.89} C_VEL
LIN {X 0,Y 98.361,Z 460.267,A -85,B 0,C 180,E1 -26729.992,E2 -26729.992} C_VEL
LIN {X 0,Y 98.236,Z 457.727,A -85,B 0,C 180,E1 -26736.152,E2 -26736.152} C_VEL
LIN {X 0,Y 98.79,Z 454.136,A -85,B 0,C 180,E1 -26742.314,E2 -26742.314} C_VEL
LIN {X 0,Y 100.222,Z 449.401,A -85,B 0,C 180,E1 -26748.385,E2 -26748.385} C_VEL
LIN {X 0,Y 103.322,Z 442.271,A -85,B 0,C 180,E1 -26755.148,E2 -26755.148} C_VEL
LIN {X 0,Y 106.793,Z 434.494,A -85,B 0,C 180,E1 -26760.654,E2 -26760.654} C_VEL
LIN {X 0,Y 110.666,Z 426.556,A -85,B 0,C 180,E1 -26764.847,E2 -26764.847} C_VEL
LIN {X 0,Y 114.864,Z 416.811,A -85,B 0,C 180,E1 -26768.827,E2 -26768.827} C_VEL
LIN {X 0,Y 118.173,Z 408.61,A -85,B 0,C 180,E1 -26771.41,E2 -26771.41} C_VEL
LIN {X 0,Y 121.782,Z 398.732,A -85,B 0,C 180,E1 -26773.815,E2 -26773.815} C_VEL
LIN {X 0,Y 125.326,Z 387.198,A -85,B 0,C 180,E1 -26775.916,E2 -26775.916} C_VEL
LIN {X 0,Y 128.393,Z 374.173,A -85,B 0,C 180,E1 -26777.628,E2 -26777.628} C_VEL
LIN {X 0,Y 130.59,Z 360.952,A -85,B 0,C 180,E1 -26778.728,E2 -26778.728} C_VEL
LIN {X 0,Y 131.43,Z 352.096,A -85,B 0,C 180,E1 -26779.242,E2 -26779.242} C_VEL
LIN {X 0,Y 131.525,Z 346.283,A -85,B 0,C 180,E1 -26779.656,E2 -26779.656} C_VEL
LIN {X 0,Y 130.498,Z 336.844,A -85,B 0,C 180,E1 -26780.821,E2 -26780.821} C_VEL
LIN {X 0,Y 129.361,Z 329.352,A -85,B 0,C 180,E1 -26781.913,E2 -26781.913} C_VEL
LIN {X 0,Y 128.641,Z 321.725,A -85,B 0,C 180,E1 -26782.86,E2 -26782.86} C_VEL
LIN {X 0,Y 128.334,Z 313.424,A -85,B 0,C 180,E1 -26783.692,E2 -26783.692} C_VEL
LIN {X 0,Y 125.055,Z 303.369,A -85,B 0,C 180,E1 -26786.292,E2 -26786.292} C_VEL
LIN {X 0,Y 122.043,Z 295.831,A -85,B 0,C 180,E1 -26788.784,E2 -26788.784} C_VEL
LIN {X 0,Y 117.195,Z 287.623,A -85,B 0,C 180,E1 -26793.001,E2 -26793.001} C_VEL
LIN {X 0,Y 113.956,Z 282.914,A -85,B 0,C 180,E1 -26796.247,E2 -26796.247} C_VEL
LIN {X 0,Y 111.577,Z 279.354,A -85,B 0,C 180,E1 -26799.008,E2 -26799.008} C_VEL
LIN {X 0,Y 109.005,Z 275.794,A -85,B 0,C 180,E1 -26802.417,E2 -26802.417} C_VEL
LIN {X 0,Y 108.188,Z 274.716,A -85,B 0,C 180,E1 -26803.628,E2 -26803.628} C_VEL
LIN {X 0,Y 105.847,Z 272.189,A -85,B 0,C 180,E1 -26807.524,E2 -26807.524} C_VEL
LIN {X 0,Y 104.841,Z 269.769,A -85,B 0,C 180,E1 -26809.865,E2 -26809.865} C_VEL
LIN {X 0,Y 102.047,Z 267.477,A -85,B 0,C 180,E1 -26818.027,E2 -26818.027} C_VEL
LIN {X 0,Y 101.606,Z 266.389,A -85,B 0,C 180,E1 -26820.991,E2 -26820.991} C_VEL
LIN {X 0,Y 101.336,Z 266.891,A -85,B 0,C 180,E1 -26828.978,E2 -26828.978} C_VEL
LIN {X 0,Y 104.702,Z 270.048,A -85,B 0,C 180,E1 -26841.666,E2 -26841.666} C_VEL
LIN {X 0,Y 106.251,Z 273.141,A -85,B 0,C 180,E1 -26845.052,E2 -26845.052} C_VEL
LIN {X 0,Y 108.681,Z 275.437,A -85,B 0,C 180,E1 -26848.856,E2 -26848.856} C_VEL
LIN {X 0,Y 111.037,Z 278.876,A -85,B 0,C 180,E1 -26852.087,E2 -26852.087} C_VEL
LIN {X 0,Y 112.383,Z 280.554,A -85,B 0,C 180,E1 -26853.69,E2 -26853.69} C_VEL
LIN {X 0,Y 115.38,Z 284.968,A -85,B 0,C 180,E1 -26856.962,E2 -26856.962} C_VEL
LIN {X 0,Y 119.225,Z 290.905,A -85,B 0,C 180,E1 -26860.57,E2 -26860.57} C_VEL
LIN {X 0,Y 123.985,Z 299.346,A -85,B 0,C 180,E1 -26864.455,E2 -26864.455} C_VEL
LIN {X 0,Y 128.444,Z 308.497,A -85,B 0,C 180,E1 -26867.681,E2 -26867.681} C_VEL
LIN {X 0,Y 129.342,Z 310.747,A -85,B 0,C 180,E1 -26868.314,E2 -26868.314} C_VEL
LIN {X 0,Y 126.124,Z 350.913,A -85,B 0,C 180,E1 -26870.181,E2 -26870.181} C_VEL
LIN {X 0,Y 124.03,Z 364.44,A -85,B 0,C 180,E1 -26871.326,E2 -26871.326} C_VEL
LIN {X 0,Y 121.2,Z 377.249,A -85,B 0,C 180,E1 -26873.026,E2 -26873.026} C_VEL
LIN {X 0,Y 118.149,Z 388.137,A -85,B 0,C 180,E1 -26875.085,E2 -26875.085} C_VEL
LIN {X 0,Y 113.957,Z 399.61,A -85,B 0,C 180,E1 -26877.876,E2 -26877.876} C_VEL
LIN {X 0,Y 109.559,Z 409.95,A -85,B 0,C 180,E1 -26881.253,E2 -26881.253} C_VEL
LIN {X 0,Y 105.203,Z 419.221,A -85,B 0,C 180,E1 -26885.332,E2 -26885.332} C_VEL
LIN {X 0,Y 100.714,Z 428.202,A -85,B 0,C 180,E1 -26890.652,E2 -26890.652} C_VEL
LIN {X 0,Y 96.884,Z 435.463,A -85,B 0,C 180,E1 -26896.373,E2 -26896.373} C_VEL
LIN {X 0,Y 94.588,Z 440.348,A -85,B 0,C 180,E1 -26901.463,E2 -26901.463} C_VEL
LIN {X 0,Y 92.577,Z 445.114,A -85,B 0,C 180,E1 -26907.833,E2 -26907.833} C_VEL
LIN {X 0,Y 91.389,Z 448.785,A -85,B 0,C 180,E1 -26914.418,E2 -26914.418} C_VEL
LIN {X 0,Y 90.932,Z 450.702,A -85,B 0,C 180,E1 -26918.9,E2 -26918.9} C_VEL
LIN {X 0,Y 90.973,Z 452.142,A -85,B 0,C 180,E1 -26923.408,E2 -26923.408} C_VEL
LIN {X 0,Y 91.472,Z 453.177,A -85,B 0,C 180,E1 -26927.905,E2 -26927.905} C_VEL
LIN {X 0,Y 93.408,Z 454.014,A -85,B 0,C 180,E1 -26935.459,E2 -26935.459} C_VEL
LIN {X 0,Y 95.664,Z 453.852,A -85,B 0,C 180,E1 -26940.954,E2 -26940.954} C_VEL
LIN {X 0,Y 100.749,Z 452.25,A -85,B 0,C 180,E1 -26948.895,E2 -26948.895} C_VEL
LIN {X 0,Y 103.927,Z 450.794,A -85,B 0,C 180,E1 -26952.556,E2 -26952.556} C_VEL
LIN {X 0,Y 109.33,Z 447.776,A -85,B 0,C 180,E1 -26957.671,E2 -26957.671} C_VEL
LIN {X 0,Y 116.535,Z 442.917,A -85,B 0,C 180,E1 -26962.908,E2 -26962.908} C_VEL
LIN {X 0,Y 124.79,Z 436.237,A -85,B 0,C 180,E1 -26967.65,E2 -26967.65} C_VEL
LIN {X 0,Y 132.681,Z 428.534,A -85,B 0,C 180,E1 -26971.361,E2 -26971.361} C_VEL
LIN {X 0,Y 140.324,Z 419.763,A -85,B 0,C 180,E1 -26974.359,E2 -26974.359} C_VEL
LIN {X 0,Y 147.247,Z 410.212,A -85,B 0,C 180,E1 -26976.75,E2 -26976.75} C_VEL
LIN {X 0,Y 153.532,Z 399.815,A -85,B 0,C 180,E1 -26978.656,E2 -26978.656} C_VEL
LIN {X 0,Y 158.729,Z 389.151,A -85,B 0,C 180,E1 -26980.198,E2 -26980.198} C_VEL
LIN {X 0,Y 163.168,Z 377.928,A -85,B 0,C 180,E1 -26981.366,E2 -26981.366} C_VEL
LIN {X 0,Y 166.881,Z 365.384,A -85,B 0,C 180,E1 -26982.292,E2 -26982.292} C_VEL
LIN {X 0,Y 169.443,Z 352.621,A -85,B 0,C 180,E1 -26982.936,E2 -26982.936} C_VEL
LIN {X 0,Y 170.307,Z 345.763,A -85,B 0,C 180,E1 -26983.21,E2 -26983.21} C_VEL
LIN {X 0,Y 167.422,Z 339.381,A -85,B 0,C 180,E1 -26986.574,E2 -26986.574} C_VEL
LIN {X 0,Y 165.332,Z 335.235,A -85,B 0,C 180,E1 -26989.456,E2 -26989.456} C_VEL
LIN {X 0,Y 163.711,Z 332.039,A -85,B 0,C 180,E1 -26992.187,E2 -26992.187} C_VEL
LIN {X 0,Y 162.21,Z 328.865,A -85,B 0,C 180,E1 -26995.472,E2 -26995.472} C_VEL
LIN {X 0,Y 160.638,Z 324.983,A -85,B 0,C 180,E1 -27001.583,E2 -27001.583} C_VEL
LIN {X 0,Y 160.595,Z 325.314,A -85,B 0,C 180,E1 -27008.81,E2 -27008.81} C_VEL
LIN {X 0,Y 161.79,Z 328.623,A -85,B 0,C 180,E1 -27013.983,E2 -27013.983} C_VEL
LIN {X 0,Y 162.484,Z 329.676,A -85,B 0,C 180,E1 -27015.684,E2 -27015.684} C_VEL
LIN {X 0,Y 164.027,Z 333.376,A -85,B 0,C 180,E1 -27018.944,E2 -27018.944} C_VEL
LIN {X 0,Y 165.648,Z 337.773,A -85,B 0,C 180,E1 -27021.724,E2 -27021.724} C_VEL
LIN {X 0,Y 167.767,Z 344.033,A -85,B 0,C 180,E1 -27024.766,E2 -27024.766} C_VEL
LIN {X 0,Y 169.855,Z 350.678,A -85,B 0,C 180,E1 -27027.363,E2 -27027.363} C_VEL
LIN {X 0,Y 168.107,Z 363.09,A -85,B 0,C 180,E1 -27027.844,E2 -27027.844} C_VEL
LIN {X 0,Y 165.176,Z 375.362,A -85,B 0,C 180,E1 -27028.484,E2 -27028.484} C_VEL
LIN {X 0,Y 161.252,Z 387.132,A -85,B 0,C 180,E1 -27029.346,E2 -27029.346} C_VEL
LIN {X 0,Y 156.021,Z 399.07,A -85,B 0,C 180,E1 -27030.516,E2 -27030.516} C_VEL
LIN {X 0,Y 150.169,Z 409.74,A -85,B 0,C 180,E1 -27031.976,E2 -27031.976} C_VEL
LIN {X 0,Y 143.752,Z 419.481,A -85,B 0,C 180,E1 -27033.784,E2 -27033.784} C_VEL
LIN {X 0,Y 136.847,Z 428.363,A -85,B 0,C 180,E1 -27036.013,E2 -27036.013} C_VEL
LIN {X 0,Y 129.018,Z 437.059,A -85,B 0,C 180,E1 -27039.08,E2 -27039.08} C_VEL
LIN {X 0,Y 121.61,Z 444.026,A -85,B 0,C 180,E1 -27042.534,E2 -27042.534} C_VEL
LIN {X 0,Y 113.609,Z 450.449,A -85,B 0,C 180,E1 -27047.115,E2 -27047.115} C_VEL
LIN {X 0,Y 108.275,Z 454.301,A -85,B 0,C 180,E1 -27051.16,E2 -27051.16} C_VEL
LIN {X 0,Y 102.39,Z 457.929,A -85,B 0,C 180,E1 -27056.688,E2 -27056.688} C_VEL
LIN {X 0,Y 96.7,Z 460.781,A -85,B 0,C 180,E1 -27064.141,E2 -27064.141} C_VEL
LIN {X 0,Y 92.951,Z 462.003,A -85,B 0,C 180,E1 -27072.389,E2 -27072.389} C_VEL
LIN {X 0,Y 91.265,Z 461.721,A -85,B 0,C 180,E1 -27081.133,E2 -27081.133} C_VEL
LIN {X 0,Y 91.144,Z 460.979,A -85,B 0,C 180,E1 -27085.57,E2 -27085.57} C_VEL
LIN {X 0,Y 91.279,Z 459.81,A -85,B 0,C 180,E1 -27089.992,E2 -27089.992} C_VEL
LIN {X 0,Y 91.155,Z 457.207,A -85,B 0,C 180,E1 -27096.632,E2 -27096.632} C_VEL
LIN {X 0,Y 91.823,Z 453.549,A -85,B 0,C 180,E1 -27103.265,E2 -27103.265} C_VEL
LIN {X 0,Y 93.472,Z 448.743,A -85,B 0,C 180,E1 -27109.766,E2 -27109.766} C_VEL
LIN {X 0,Y 96.34,Z 442.668,A -85,B 0,C 180,E1 -27115.946,E2 -27115.946} C_VEL
LIN {X 0,Y 100.002,Z 435.069,A -85,B 0,C 180,E1 -27121.792,E2 -27121.792} C_VEL
LIN {X 0,Y 104.022,Z 427.33,A -85,B 0,C 180,E1 -27126.226,E2 -27126.226} C_VEL
LIN {X 0,Y 108.437,Z 417.863,A -85,B 0,C 180,E1 -27130.386,E2 -27130.386} C_VEL
LIN {X 0,Y 111.328,Z 411.088,A -85,B 0,C 180,E1 -27132.722,E2 -27132.722} C_VEL
LIN {X 0,Y 115.647,Z 400.4,A -85,B 0,C 180,E1 -27135.551,E2 -27135.551} C_VEL
LIN {X 0,Y 119.585,Z 388.413,A -85,B 0,C 180,E1 -27137.884,E2 -27137.884} C_VEL
LIN {X 0,Y 122.779,Z 375.898,A -85,B 0,C 180,E1 -27139.627,E2 -27139.627} C_VEL
LIN {X 0,Y 125.224,Z 362.98,A -85,B 0,C 180,E1 -27140.807,E2 -27140.807} C_VEL
LIN {X 0,Y 126.722,Z 348.107,A -85,B 0,C 180,E1 -27141.638,E2 -27141.638} C_VEL
LIN {X 0,Y 128.656,Z 322.104,A -85,B 0,C 180,E1 -27142.822,E2 -27142.822} C_VEL
LIN {X 0,Y 128.641,Z 321.725,A -85,B 0,C 180,E1 -27142.86,E2 -27142.86} C_VEL
LIN {X 0,Y 128.07,Z 318.771,A -85,B 0,C 180,E1 -27143.381,E2 -27143.381} C_VEL
LIN {X 0,Y 126.322,Z 315.376,A -85,B 0,C 180,E1 -27144.554,E2 -27144.554} C_VEL
LIN {X 0,Y 122.004,Z 309.536,A -85,B 0,C 180,E1 -27147.496,E2 -27147.496} C_VEL
LIN {X 0,Y 120.695,Z 306.404,A -85,B 0,C 180,E1 -27148.603,E2 -27148.603} C_VEL
LIN {X 0,Y 118.422,Z 300.49,A -85,B 0,C 180,E1 -27150.708,E2 -27150.708} C_VEL
LIN {X 0,Y 114.436,Z 293.366,A -85,B 0,C 180,E1 -27154.539,E2 -27154.539} C_VEL
LIN {X 0,Y 111.218,Z 288.51,A -85,B 0,C 180,E1 -27158.086,E2 -27158.086} C_VEL
LIN {X 0,Y 109.192,Z 285.38,A -85,B 0,C 180,E1 -27160.679,E2 -27160.679} C_VEL
LIN {X 0,Y 106.511,Z 281.361,A -85,B 0,C 180,E1 -27164.697,E2 -27164.697} C_VEL
LIN {X 0,Y 104.196,Z 278.586,A -85,B 0,C 180,E1 -27168.942,E2 -27168.942} C_VEL
LIN {X 0,Y 103.331,Z 276.502,A -85,B 0,C 180,E1 -27171.167,E2 -27171.167} C_VEL
LIN {X 0,Y 101.015,Z 274.382,A -85,B 0,C 180,E1 -27178.755,E2 -27178.755} C_VEL
LIN {X 0,Y 100.725,Z 273.442,A -85,B 0,C 180,E1 -27181,E2 -27181} C_VEL
LIN {X 0,Y 100.462,Z 273.979,A -85,B 0,C 180,E1 -27189.057,E2 -27189.057} C_VEL
LIN {X 0,Y 103.274,Z 276.87,A -85,B 0,C 180,E1 -27200.54,E2 -27200.54} C_VEL
LIN {X 0,Y 105.075,Z 280.228,A -85,B 0,C 180,E1 -27204.657,E2 -27204.657} C_VEL
LIN {X 0,Y 106.834,Z 281.947,A -85,B 0,C 180,E1 -27207.585,E2 -27207.585} C_VEL
LIN {X 0,Y 109.457,Z 285.74,A -85,B 0,C 180,E1 -27211.402,E2 -27211.402} C_VEL
LIN {X 0,Y 112.885,Z 291.029,A -85,B 0,C 180,E1 -27215.548,E2 -27215.548} C_VEL
LIN {X 0,Y 116.211,Z 296.439,A -85,B 0,C 180,E1 -27218.961,E2 -27218.961} C_VEL
LIN {X 0,Y 120.683,Z 304.775,A -85,B 0,C 180,E1 -27222.955,E2 -27222.955} C_VEL
LIN {X 0,Y 124.504,Z 313.175,A -85,B 0,C 180,E1 -27226.004,E2 -27226.004} C_VEL
LIN {X 0,Y 121.318,Z 350.915,A -85,B 0,C 180,E1 -27227.759,E2 -27227.759} C_VEL
LIN {X 0,Y 119.112,Z 364.673,A -85,B 0,C 180,E1 -27228.929,E2 -27228.929} C_VEL
LIN {X 0,Y 116.218,Z 377.222,A -85,B 0,C 180,E1 -27230.596,E2 -27230.596} C_VEL
LIN {X 0,Y 112.985,Z 388.187,A -85,B 0,C 180,E1 -27232.677,E2 -27232.677} C_VEL
LIN {X 0,Y 108.565,Z 399.709,A -85,B 0,C 180,E1 -27235.51,E2 -27235.51} C_VEL
LIN {X 0,Y 103.893,Z 410.09,A -85,B 0,C 180,E1 -27238.961,E2 -27238.961} C_VEL
LIN {X 0,Y 99.702,Z 418.56,A -85,B 0,C 180,E1 -27242.742,E2 -27242.742} C_VEL
LIN {X 0,Y 94.783,Z 427.734,A -85,B 0,C 180,E1 -27248.249,E2 -27248.249} C_VEL
LIN {X 0,Y 90.584,Z 435.133,A -85,B 0,C 180,E1 -27254.254,E2 -27254.254} C_VEL
LIN {X 0,Y 87.575,Z 441.049,A -85,B 0,C 180,E1 -27260.774,E2 -27260.774} C_VEL
LIN {X 0,Y 85.468,Z 445.737,A -85,B 0,C 180,E1 -27267.653,E2 -27267.653} C_VEL
LIN {X 0,Y 84.216,Z 449.339,A -85,B 0,C 180,E1 -27274.796,E2 -27274.796} C_VEL
LIN {X 0,Y 83.812,Z 451.195,A -85,B 0,C 180,E1 -27279.663,E2 -27279.663} C_VEL
LIN {X 0,Y 83.956,Z 452.593,A -85,B 0,C 180,E1 -27284.552,E2 -27284.552} C_VEL
LIN {X 0,Y 85.769,Z 454.204,A -85,B 0,C 180,E1 -27294.194,E2 -27294.194} C_VEL
LIN {X 0,Y 87.392,Z 454.375,A -85,B 0,C 180,E1 -27298.856,E2 -27298.856} C_VEL
LIN {X 0,Y 92.092,Z 453.502,A -85,B 0,C 180,E1 -27307.633,E2 -27307.633} C_VEL
LIN {X 0,Y 96.685,Z 451.819,A -85,B 0,C 180,E1 -27313.372,E2 -27313.372} C_VEL
LIN {X 0,Y 104.554,Z 447.848,A -85,B 0,C 180,E1 -27320.63,E2 -27320.63} C_VEL
LIN {X 0,Y 111.63,Z 443.362,A -85,B 0,C 180,E1 -27325.484,E2 -27325.484} C_VEL
LIN {X 0,Y 119.756,Z 437.186,A -85,B 0,C 180,E1 -27329.956,E2 -27329.956} C_VEL
LIN {X 0,Y 127.469,Z 430.194,A -85,B 0,C 180,E1 -27333.444,E2 -27333.444} C_VEL
LIN {X 0,Y 134.494,Z 422.717,A -85,B 0,C 180,E1 -27336.131,E2 -27336.131} C_VEL
LIN {X 0,Y 141.621,Z 413.775,A -85,B 0,C 180,E1 -27338.51,E2 -27338.51} C_VEL
LIN {X 0,Y 148.356,Z 403.709,A -85,B 0,C 180,E1 -27340.476,E2 -27340.476} C_VEL
LIN {X 0,Y 154.158,Z 392.992,A -85,B 0,C 180,E1 -27342.114,E2 -27342.114} C_VEL
LIN {X 0,Y 159.068,Z 381.652,A -85,B 0,C 180,E1 -27343.374,E2 -27343.374} C_VEL
LIN {X 0,Y 163.175,Z 369.447,A -85,B 0,C 180,E1 -27344.311,E2 -27344.311} C_VEL
LIN {X 0,Y 166.228,Z 356.379,A -85,B 0,C 180,E1 -27345.053,E2 -27345.053} C_VEL
LIN {X 0,Y 167.274,Z 349.564,A -85,B 0,C 180,E1 -27345.336,E2 -27345.336} C_VEL
LIN {X 0,Y 164.784,Z 343.739,A -85,B 0,C 180,E1 -27348.802,E2 -27348.802} C_VEL
LIN {X 0,Y 162.427,Z 338.766,A -85,B 0,C 180,E1 -27352.851,E2 -27352.851} C_VEL
LIN {X 0,Y 161.024,Z 335.666,A -85,B 0,C 180,E1 -27356.175,E2 -27356.175} C_VEL
LIN {X 0,Y 159.713,Z 332.01,A -85,B 0,C 180,E1 -27361.891,E2 -27361.891} C_VEL
LIN {X 0,Y 159.642,Z 332.22,A -85,B 0,C 180,E1 -27368.226,E2 -27368.226} C_VEL
LIN {X 0,Y 160.84,Z 335.667,A -85,B 0,C 180,E1 -27373.825,E2 -27373.825} C_VEL
LIN {X 0,Y 161.461,Z 336.888,A -85,B 0,C 180,E1 -27375.462,E2 -27375.462} C_VEL
LIN {X 0,Y 162.646,Z 340.039,A -85,B 0,C 180,E1 -27378.161,E2 -27378.161} C_VEL
LIN {X 0,Y 164.211,Z 344.713,A -85,B 0,C 180,E1 -27381.086,E2 -27381.086} C_VEL
LIN {X 0,Y 166.244,Z 351.476,A -85,B 0,C 180,E1 -27384.259,E2 -27384.259} C_VEL
LIN {X 0,Y 166.876,Z 353.836,A -85,B 0,C 180,E1 -27385.207,E2 -27385.207} C_VEL
LIN {X 0,Y 165.402,Z 363.216,A -85,B 0,C 180,E1 -27385.59,E2 -27385.59} C_VEL
LIN {X 0,Y 162.297,Z 375.712,A -85,B 0,C 180,E1 -27386.224,E2 -27386.224} C_VEL
LIN {X 0,Y 157.915,Z 388.246,A -85,B 0,C 180,E1 -27387.115,E2 -27387.115} C_VEL
LIN {X 0,Y 152.55,Z 399.794,A -85,B 0,C 180,E1 -27388.226,E2 -27388.226} C_VEL
LIN {X 0,Y 146.552,Z 410.266,A -85,B 0,C 180,E1 -27389.634,E2 -27389.634} C_VEL
LIN {X 0,Y 139.947,Z 419.862,A -85,B 0,C 180,E1 -27391.38,E2 -27391.38} C_VEL
LIN {X 0,Y 132.805,Z 428.629,A -85,B 0,C 180,E1 -27393.54,E2 -27393.54} C_VEL
LIN {X 0,Y 124.668,Z 437.188,A -85,B 0,C 180,E1 -27396.548,E2 -27396.548} C_VEL
LIN {X 0,Y 116.918,Z 444.066,A -85,B 0,C 180,E1 -27399.964,E2 -27399.964} C_VEL
LIN {X 0,Y 108.515,Z 450.415,A -85,B 0,C 180,E1 -27404.564,E2 -27404.564} C_VEL
LIN {X 0,Y 102.376,Z 454.482,A -85,B 0,C 180,E1 -27409.037,E2 -27409.037} C_VEL
LIN {X 0,Y 96.527,Z 457.763,A -85,B 0,C 180,E1 -27414.37,E2 -27414.37} C_VEL
LIN {X 0,Y 93.202,Z 459.358,A -85,B 0,C 180,E1 -27418.134,E2 -27418.134} C_VEL
LIN {X 0,Y 90.336,Z 460.532,A -85,B 0,C 180,E1 -27422.167,E2 -27422.167} C_VEL
LIN {X 0,Y 86.188,Z 461.689,A -85,B 0,C 180,E1 -27430.956,E2 -27430.956} C_VEL
LIN {X 0,Y 84.242,Z 461.341,A -85,B 0,C 180,E1 -27440.387,E2 -27440.387} C_VEL
LIN {X 0,Y 84.059,Z 460.549,A -85,B 0,C 180,E1 -27445.195,E2 -27445.195} C_VEL
LIN {X 0,Y 84.188,Z 459.351,A -85,B 0,C 180,E1 -27449.991,E2 -27449.991} C_VEL
LIN {X 0,Y 84.098,Z 456.685,A -85,B 0,C 180,E1 -27457.191,E2 -27457.191} C_VEL
LIN {X 0,Y 84.898,Z 452.959,A -85,B 0,C 180,E1 -27464.369,E2 -27464.369} C_VEL
LIN {X 0,Y 86.769,Z 448.081,A -85,B 0,C 180,E1 -27471.364,E2 -27471.364} C_VEL
LIN {X 0,Y 89.957,Z 441.928,A -85,B 0,C 180,E1 -27477.941,E2 -27477.941} C_VEL
LIN {X 0,Y 93.773,Z 434.6,A -85,B 0,C 180,E1 -27483.842,E2 -27483.842} C_VEL
LIN {X 0,Y 98.338,Z 426.388,A -85,B 0,C 180,E1 -27488.692,E2 -27488.692} C_VEL
LIN {X 0,Y 103.069,Z 416.742,A -85,B 0,C 180,E1 -27492.975,E2 -27492.975} C_VEL
LIN {X 0,Y 106.759,Z 408.663,A -85,B 0,C 180,E1 -27495.701,E2 -27495.701} C_VEL
LIN {X 0,Y 110.747,Z 398.945,A -85,B 0,C 180,E1 -27498.199,E2 -27498.199} C_VEL
LIN {X 0,Y 114.925,Z 386.626,A -85,B 0,C 180,E1 -27500.522,E2 -27500.522} C_VEL
LIN {X 0,Y 118.116,Z 374.417,A -85,B 0,C 180,E1 -27502.166,E2 -27502.166} C_VEL
LIN {X 0,Y 120.512,Z 361.55,A -85,B 0,C 180,E1 -27503.3,E2 -27503.3} C_VEL
LIN {X 0,Y 122.177,Z 345.023,A -85,B 0,C 180,E1 -27504.171,E2 -27504.171} C_VEL
LIN {X 0,Y 123.902,Z 322.831,A -85,B 0,C 180,E1 -27505.197,E2 -27505.197} C_VEL
LIN {X 0,Y 123.735,Z 316.169,A -85,B 0,C 180,E1 -27505.883,E2 -27505.883} C_VEL
LIN {X 0,Y 121.104,Z 307.511,A -85,B 0,C 180,E1 -27508.239,E2 -27508.239} C_VEL
LIN {X 0,Y 120.695,Z 306.404,A -85,B 0,C 180,E1 -27508.603,E2 -27508.603} C_VEL
LIN {X 0,Y 119.614,Z 304.097,A -85,B 0,C 180,E1 -27509.53,E2 -27509.53} C_VEL
LIN {X 0,Y 117.437,Z 302.095,A -85,B 0,C 180,E1 -27511.233,E2 -27511.233} C_VEL
LIN {X 0,Y 112.051,Z 299.253,A -85,B 0,C 180,E1 -27515.872,E2 -27515.872} C_VEL
LIN {X 0,Y 110.988,Z 297.986,A -85,B 0,C 180,E1 -27517.02,E2 -27517.02} C_VEL
LIN {X 0,Y 108.423,Z 293.751,A -85,B 0,C 180,E1 -27520.259,E2 -27520.259} C_VEL
LIN {X 0,Y 106.983,Z 291.419,A -85,B 0,C 180,E1 -27522.313,E2 -27522.313} C_VEL
LIN {X 0,Y 104.721,Z 287.888,A -85,B 0,C 180,E1 -27526.052,E2 -27526.052} C_VEL
LIN {X 0,Y 102.508,Z 284.754,A -85,B 0,C 180,E1 -27530.676,E2 -27530.676} C_VEL
LIN {X 0,Y 101.898,Z 283.279,A -85,B 0,C 180,E1 -27532.445,E2 -27532.445} C_VEL
LIN {X 0,Y 99.904,Z 280.997,A -85,B 0,C 180,E1 -27540.252,E2 -27540.252} C_VEL
LIN {X 0,Y 99.723,Z 280.456,A -85,B 0,C 180,E1 -27542.02,E2 -27542.02} C_VEL
LIN {X 0,Y 99.684,Z 281.229,A -85,B 0,C 180,E1 -27550.152,E2 -27550.152} C_VEL
LIN {X 0,Y 101.955,Z 283.83,A -85,B 0,C 180,E1 -27559.579,E2 -27559.579} C_VEL
LIN {X 0,Y 103.766,Z 287.123,A -85,B 0,C 180,E1 -27563.978,E2 -27563.978} C_VEL
LIN {X 0,Y 105.219,Z 288.755,A -85,B 0,C 180,E1 -27566.588,E2 -27566.588} C_VEL
LIN {X 0,Y 108.064,Z 293.157,A -85,B 0,C 180,E1 -27570.978,E2 -27570.978} C_VEL
LIN {X 0,Y 110.683,Z 297.45,A -85,B 0,C 180,E1 -27574.336,E2 -27574.336} C_VEL
LIN {X 0,Y 113.856,Z 303.117,A -85,B 0,C 180,E1 -27577.871,E2 -27577.871} C_VEL
LIN {X 0,Y 117.304,Z 309.908,A -85,B 0,C 180,E1 -27581.227,E2 -27581.227} C_VEL
LIN {X 0,Y 119.87,Z 315.732,A -85,B 0,C 180,E1 -27583.514,E2 -27583.514} C_VEL
LIN {X 0,Y 116.628,Z 351.866,A -85,B 0,C 180,E1 -27585.213,E2 -27585.213} C_VEL
LIN {X 0,Y 114.336,Z 365.323,A -85,B 0,C 180,E1 -27586.372,E2 -27586.372} C_VEL
LIN {X 0,Y 111.161,Z 378.196,A -85,B 0,C 180,E1 -27588.117,E2 -27588.117} C_VEL
LIN {X 0,Y 107.436,Z 389.82,A -85,B 0,C 180,E1 -27590.386,E2 -27590.386} C_VEL
LIN {X 0,Y 102.826,Z 401.096,A -85,B 0,C 180,E1 -27593.283,E2 -27593.283} C_VEL
LIN {X 0,Y 97.877,Z 411.273,A -85,B 0,C 180,E1 -27596.817,E2 -27596.817} C_VEL
LIN {X 0,Y 92.509,Z 421.217,A -85,B 0,C 180,E1 -27601.665,E2 -27601.665} C_VEL
LIN {X 0,Y 87.418,Z 429.978,A -85,B 0,C 180,E1 -27607.562,E2 -27607.562} C_VEL
LIN {X 0,Y 83.176,Z 436.983,A -85,B 0,C 180,E1 -27614.072,E2 -27614.072} C_VEL
LIN {X 0,Y 79.66,Z 443.391,A -85,B 0,C 180,E1 -27622.406,E2 -27622.406} C_VEL
LIN {X 0,Y 77.828,Z 447.623,A -85,B 0,C 180,E1 -27630.01,E2 -27630.01} C_VEL
LIN {X 0,Y 77.051,Z 449.891,A -85,B 0,C 180,E1 -27635.243,E2 -27635.243} C_VEL
LIN {X 0,Y 76.698,Z 451.68,A -85,B 0,C 180,E1 -27640.569,E2 -27640.569} C_VEL
LIN {X 0,Y 76.959,Z 453.045,A -85,B 0,C 180,E1 -27645.909,E2 -27645.909} C_VEL
LIN {X 0,Y 77.791,Z 454.014,A -85,B 0,C 180,E1 -27651.193,E2 -27651.193} C_VEL
LIN {X 0,Y 79.887,Z 454.655,A -85,B 0,C 180,E1 -27658.387,E2 -27658.387} C_VEL
LIN {X 0,Y 83.479,Z 454.422,A -85,B 0,C 180,E1 -27666.116,E2 -27666.116} C_VEL
LIN {X 0,Y 86.432,Z 453.753,A -85,B 0,C 180,E1 -27670.586,E2 -27670.586} C_VEL
LIN {X 0,Y 90.955,Z 452.213,A -85,B 0,C 180,E1 -27675.939,E2 -27675.939} C_VEL
LIN {X 0,Y 97.847,Z 449.105,A -85,B 0,C 180,E1 -27682.2,E2 -27682.2} C_VEL
LIN {X 0,Y 104.626,Z 445.292,A -85,B 0,C 180,E1 -27686.905,E2 -27686.905} C_VEL
LIN {X 0,Y 112.298,Z 440.126,A -85,B 0,C 180,E1 -27691.187,E2 -27691.187} C_VEL
LIN {X 0,Y 120.365,Z 433.655,A -85,B 0,C 180,E1 -27694.83,E2 -27694.83} C_VEL
LIN {X 0,Y 128.825,Z 425.51,A -85,B 0,C 180,E1 -27698.04,E2 -27698.04} C_VEL
LIN {X 0,Y 136.143,Z 417.147,A -85,B 0,C 180,E1 -27700.409,E2 -27700.409} C_VEL
LIN {X 0,Y 143.348,Z 407.33,A -85,B 0,C 180,E1 -27702.454,E2 -27702.454} C_VEL
LIN {X 0,Y 149.771,Z 396.509,A -85,B 0,C 180,E1 -27704.145,E2 -27704.145} C_VEL
LIN {X 0,Y 155.165,Z 385.154,A -85,B 0,C 180,E1 -27705.499,E2 -27705.499} C_VEL
LIN {X 0,Y 159.828,Z 372.72,A -85,B 0,C 180,E1 -27706.474,E2 -27706.474} C_VEL
LIN {X 0,Y 163.311,Z 359.231,A -85,B 0,C 180,E1 -27707.26,E2 -27707.26} C_VEL
LIN {X 0,Y 164.362,Z 353.589,A -85,B 0,C 180,E1 -27707.498,E2 -27707.498} C_VEL
LIN {X 0,Y 162.584,Z 348.783,A -85,B 0,C 180,E1 -27710.671,E2 -27710.671} C_VEL
LIN {X 0,Y 160.996,Z 345.166,A -85,B 0,C 180,E1 -27713.892,E2 -27713.892} C_VEL
LIN {X 0,Y 159.884,Z 342.432,A -85,B 0,C 180,E1 -27716.85,E2 -27716.85} C_VEL
LIN {X 0,Y 158.751,Z 338.985,A -85,B 0,C 180,E1 -27722.537,E2 -27722.537} C_VEL
LIN {X 0,Y 158.739,Z 339.367,A -85,B 0,C 180,E1 -27728.113,E2 -27728.113} C_VEL
LIN {X 0,Y 159.78,Z 342.561,A -85,B 0,C 180,E1 -27733.351,E2 -27733.351} C_VEL
LIN {X 0,Y 160.385,Z 343.915,A -85,B 0,C 180,E1 -27735.08,E2 -27735.08} C_VEL
LIN {X 0,Y 161.405,Z 347.034,A -85,B 0,C 180,E1 -27737.61,E2 -27737.61} C_VEL
LIN {X 0,Y 162.651,Z 351.298,A -85,B 0,C 180,E1 -27740.223,E2 -27740.223} C_VEL
LIN {X 0,Y 164.067,Z 357.303,A -85,B 0,C 180,E1 -27743.037,E2 -27743.037} C_VEL
LIN {X 0,Y 161.202,Z 370.724,A -85,B 0,C 180,E1 -27743.583,E2 -27743.583} C_VEL
LIN {X 0,Y 157.253,Z 383.251,A -85,B 0,C 180,E1 -27744.346,E2 -27744.346} C_VEL
LIN {X 0,Y 151.675,Z 395.998,A -85,B 0,C 180,E1 -27745.372,E2 -27745.372} C_VEL
LIN {X 0,Y 145.47,Z 407.208,A -85,B 0,C 180,E1 -27746.647,E2 -27746.647} C_VEL
LIN {X 0,Y 138.676,Z 417.318,A -85,B 0,C 180,E1 -27748.29,E2 -27748.29} C_VEL
LIN {X 0,Y 130.439,Z 427.27,A -85,B 0,C 180,E1 -27750.448,E2 -27750.448} C_VEL
LIN {X 0,Y 121.983,Z 436.043,A -85,B 0,C 180,E1 -27753.339,E2 -27753.339} C_VEL
LIN {X 0,Y 113.815,Z 443.093,A -85,B 0,C 180,E1 -27756.604,E2 -27756.604} C_VEL
LIN {X 0,Y 106.084,Z 448.755,A -85,B 0,C 180,E1 -27760.366,E2 -27760.366} C_VEL
LIN {X 0,Y 99.023,Z 453.244,A -85,B 0,C 180,E1 -27764.782,E2 -27764.782} C_VEL
LIN {X 0,Y 94.77,Z 455.63,A -85,B 0,C 180,E1 -27768.126,E2 -27768.126} C_VEL
LIN {X 0,Y 90.841,Z 457.598,A -85,B 0,C 180,E1 -27771.756,E2 -27771.756} C_VEL
LIN {X 0,Y 87.225,Z 459.156,A -85,B 0,C 180,E1 -27775.659,E2 -27775.659} C_VEL
LIN {X 0,Y 81.458,Z 461.01,A -85,B 0,C 180,E1 -27784.437,E2 -27784.437} C_VEL
LIN {X 0,Y 78.077,Z 461.365,A -85,B 0,C 180,E1 -27794.325,E2 -27794.325} C_VEL
LIN {X 0,Y 77.229,Z 460.944,A -85,B 0,C 180,E1 -27799.505,E2 -27799.505} C_VEL
LIN {X 0,Y 76.976,Z 460.119,A -85,B 0,C 180,E1 -27804.752,E2 -27804.752} C_VEL
LIN {X 0,Y 77.104,Z 458.892,A -85,B 0,C 180,E1 -27809.99,E2 -27809.99} C_VEL
LIN {X 0,Y 77.048,Z 456.162,A -85,B 0,C 180,E1 -27817.853,E2 -27817.853} C_VEL
LIN {X 0,Y 77.99,Z 452.368,A -85,B 0,C 180,E1 -27825.673,E2 -27825.673} C_VEL
LIN {X 0,Y 80.158,Z 447.419,A -85,B 0,C 180,E1 -27833.225,E2 -27833.225} C_VEL
LIN {X 0,Y 83.659,Z 441.183,A -85,B 0,C 180,E1 -27840.254,E2 -27840.254} C_VEL
LIN {X 0,Y 87.446,Z 434.556,A -85,B 0,C 180,E1 -27845.855,E2 -27845.855} C_VEL
LIN {X 0,Y 92.845,Z 425.404,A -85,B 0,C 180,E1 -27851.463,E2 -27851.463} C_VEL
LIN {X 0,Y 97.89,Z 415.611,A -85,B 0,C 180,E1 -27855.869,E2 -27855.869} C_VEL
LIN {X 0,Y 103.115,Z 404.787,A -85,B 0,C 180,E1 -27859.292,E2 -27859.292} C_VEL
LIN {X 0,Y 107.365,Z 394.24,A -85,B 0,C 180,E1 -27861.749,E2 -27861.749} C_VEL
LIN {X 0,Y 111.469,Z 381.509,A -85,B 0,C 180,E1 -27863.864,E2 -27863.864} C_VEL
LIN {X 0,Y 114.664,Z 368.392,A -85,B 0,C 180,E1 -27865.337,E2 -27865.337} C_VEL
LIN {X 0,Y 116.647,Z 355.215,A -85,B 0,C 180,E1 -27866.302,E2 -27866.302} C_VEL
LIN {X 0,Y 119.374,Z 323.591,A -85,B 0,C 180,E1 -27867.756,E2 -27867.756} C_VEL
LIN {X 0,Y 119.252,Z 318.516,A -85,B 0,C 180,E1 -27868.328,E2 -27868.328} C_VEL
LIN {X 0,Y 116.959,Z 310.681,A -85,B 0,C 180,E1 -27870.657,E2 -27870.657} C_VEL
LIN {X 0,Y 115.086,Z 305.414,A -85,B 0,C 180,E1 -27872.611,E2 -27872.611} C_VEL
LIN {X 0,Y 111.459,Z 298.704,A -85,B 0,C 180,E1 -27876.483,E2 -27876.483} C_VEL
LIN {X 0,Y 110.988,Z 297.986,A -85,B 0,C 180,E1 -27877.02,E2 -27877.02} C_VEL
LIN {X 0,Y 109.498,Z 296.396,A -85,B 0,C 180,E1 -27878.721,E2 -27878.721} C_VEL
LIN {X 0,Y 106.778,Z 295.478,A -85,B 0,C 180,E1 -27881.893,E2 -27881.893} C_VEL
LIN {X 0,Y 103.803,Z 294.957,A -85,B 0,C 180,E1 -27886.036,E2 -27886.036} C_VEL
LIN {X 0,Y 103.006,Z 294.381,A -85,B 0,C 180,E1 -27887.438,E2 -27887.438} C_VEL
LIN {X 0,Y 100.947,Z 290.994,A -85,B 0,C 180,E1 -27892.374,E2 -27892.374} C_VEL
LIN {X 0,Y 100.613,Z 290.123,A -85,B 0,C 180,E1 -27893.483,E2 -27893.483} C_VEL
LIN {X 0,Y 98.887,Z 287.671,A -85,B 0,C 180,E1 -27901.528,E2 -27901.528} C_VEL
LIN {X 0,Y 98.626,Z 287.85,A -85,B 0,C 180,E1 -27907.263,E2 -27907.263} C_VEL
LIN {X 0,Y 100.529,Z 290.382,A -85,B 0,C 180,E1 -27918.106,E2 -27918.106} C_VEL
LIN {X 0,Y 102.595,Z 294.143,A -85,B 0,C 180,E1 -27923.53,E2 -27923.53} C_VEL
LIN {X 0,Y 103.473,Z 295.23,A -85,B 0,C 180,E1 -27925.234,E2 -27925.234} C_VEL
LIN {X 0,Y 106.117,Z 299.621,A -85,B 0,C 180,E1 -27929.715,E2 -27929.715} C_VEL
LIN {X 0,Y 109.226,Z 305.043,A -85,B 0,C 180,E1 -27933.949,E2 -27933.949} C_VEL
LIN {X 0,Y 113.166,Z 313.076,A -85,B 0,C 180,E1 -27938.488,E2 -27938.488} C_VEL
LIN {X 0,Y 115.456,Z 318.346,A -85,B 0,C 180,E1 -27940.82,E2 -27940.82} C_VEL
LIN {X 0,Y 112.304,Z 351.94,A -85,B 0,C 180,E1 -27942.395,E2 -27942.395} C_VEL
LIN {X 0,Y 109.877,Z 365.638,A -85,B 0,C 180,E1 -27943.565,E2 -27943.565} C_VEL
LIN {X 0,Y 106.645,Z 378.176,A -85,B 0,C 180,E1 -27945.242,E2 -27945.242} C_VEL
LIN {X 0,Y 102.709,Z 389.87,A -85,B 0,C 180,E1 -27947.506,E2 -27947.506} C_VEL
LIN {X 0,Y 97.841,Z 401.196,A -85,B 0,C 180,E1 -27950.409,E2 -27950.409} C_VEL
LIN {X 0,Y 92.58,Z 411.425,A -85,B 0,C 180,E1 -27953.976,E2 -27953.976} C_VEL
LIN {X 0,Y 87.346,Z 420.585,A -85,B 0,C 180,E1 -27958.48,E2 -27958.48} C_VEL
LIN {X 0,Y 81.754,Z 429.509,A -85,B 0,C 180,E1 -27964.556,E2 -27964.556} C_VEL
LIN {X 0,Y 77.026,Z 436.705,A -85,B 0,C 180,E1 -27971.389,E2 -27971.389} C_VEL
LIN {X 0,Y 73.574,Z 442.427,A -85,B 0,C 180,E1 -27978.998,E2 -27978.998} C_VEL
LIN {X 0,Y 71.24,Z 446.95,A -85,B 0,C 180,E1 -27987.184,E2 -27987.184} C_VEL
LIN {X 0,Y 69.88,Z 450.423,A -85,B 0,C 180,E1 -27995.782,E2 -27995.782} C_VEL
LIN {X 0,Y 69.623,Z 452.164,A -85,B 0,C 180,E1 -28001.657,E2 -28001.657} C_VEL
LIN {X 0,Y 70.014,Z 453.498,A -85,B 0,C 180,E1 -28007.536,E2 -28007.536} C_VEL
LIN {X 0,Y 71.084,Z 454.431,A -85,B 0,C 180,E1 -28013.305,E2 -28013.305} C_VEL
LIN {X 0,Y 73.228,Z 454.976,A -85,B 0,C 180,E1 -28020.256,E2 -28020.256} C_VEL
LIN {X 0,Y 77.711,Z 454.706,A -85,B 0,C 180,E1 -28029.284,E2 -28029.284} C_VEL
LIN {X 0,Y 81.019,Z 453.997,A -85,B 0,C 180,E1 -28033.952,E2 -28033.952} C_VEL
LIN {X 0,Y 85.376,Z 452.622,A -85,B 0,C 180,E1 -28038.81,E2 -28038.81} C_VEL
LIN {X 0,Y 93.546,Z 449.215,A -85,B 0,C 180,E1 -28045.738,E2 -28045.738} C_VEL
LIN {X 0,Y 102.549,Z 444.275,A -85,B 0,C 180,E1 -28051.331,E2 -28051.331} C_VEL
LIN {X 0,Y 111.748,Z 438.02,A -85,B 0,C 180,E1 -28055.777,E2 -28055.777} C_VEL
LIN {X 0,Y 120.342,Z 430.943,A -85,B 0,C 180,E1 -28059.134,E2 -28059.134} C_VEL
LIN {X 0,Y 129.291,Z 422.006,A -85,B 0,C 180,E1 -28062.04,E2 -28062.04} C_VEL
LIN {X 0,Y 136.953,Z 412.792,A -85,B 0,C 180,E1 -28064.195,E2 -28064.195} C_VEL
LIN {X 0,Y 143.745,Z 402.973,A -85,B 0,C 180,E1 -28065.85,E2 -28065.85} C_VEL
LIN {X 0,Y 150.315,Z 391.001,A -85,B 0,C 180,E1 -28067.424,E2 -28067.424} C_VEL
LIN {X 0,Y 155.021,Z 380.301,A -85,B 0,C 180,E1 -28068.4,E2 -28068.4} C_VEL
LIN {X 0,Y 159.179,Z 367.951,A -85,B 0,C 180,E1 -28069.214,E2 -28069.214} C_VEL
LIN {X 0,Y 161.585,Z 357.631,A -85,B 0,C 180,E1 -28069.787,E2 -28069.787} C_VEL
LIN {X 0,Y 159.878,Z 352.33,A -85,B 0,C 180,E1 -28074.007,E2 -28074.007} C_VEL
LIN {X 0,Y 158.739,Z 349.244,A -85,B 0,C 180,E1 -28077.462,E2 -28077.462} C_VEL
LIN {X 0,Y 157.873,Z 346.061,A -85,B 0,C 180,E1 -28082.551,E2 -28082.551} C_VEL
LIN {X 0,Y 157.835,Z 346.539,A -85,B 0,C 180,E1 -28087.998,E2 -28087.998} C_VEL
LIN {X 0,Y 159.086,Z 350.304,A -85,B 0,C 180,E1 -28094.06,E2 -28094.06} C_VEL
LIN {X 0,Y 159.943,Z 353.463,A -85,B 0,C 180,E1 -28096.677,E2 -28096.677} C_VEL
LIN {X 0,Y 160.94,Z 358.251,A -85,B 0,C 180,E1 -28099.532,E2 -28099.532} C_VEL
LIN {X 0,Y 161.372,Z 360.728,A -85,B 0,C 180,E1 -28100.746,E2 -28100.746} C_VEL
LIN {X 0,Y 158.387,Z 373.007,A -85,B 0,C 180,E1 -28101.281,E2 -28101.281} C_VEL
LIN {X 0,Y 154.056,Z 385.433,A -85,B 0,C 180,E1 -28102.031,E2 -28102.031} C_VEL
LIN {X 0,Y 148.788,Z 396.829,A -85,B 0,C 180,E1 -28102.916,E2 -28102.916} C_VEL
LIN {X 0,Y 142.439,Z 407.803,A -85,B 0,C 180,E1 -28104.105,E2 -28104.105} C_VEL
LIN {X 0,Y 134.692,Z 418.676,A -85,B 0,C 180,E1 -28105.831,E2 -28105.831} C_VEL
LIN {X 0,Y 127.001,Z 427.534,A -85,B 0,C 180,E1 -28107.696,E2 -28107.696} C_VEL
LIN {X 0,Y 118.228,Z 436.193,A -85,B 0,C 180,E1 -28110.462,E2 -28110.462} C_VEL
LIN {X 0,Y 109.728,Z 443.133,A -85,B 0,C 180,E1 -28113.625,E2 -28113.625} C_VEL
LIN {X 0,Y 101.618,Z 448.721,A -85,B 0,C 180,E1 -28117.307,E2 -28117.307} C_VEL
LIN {X 0,Y 94.139,Z 453.141,A -85,B 0,C 180,E1 -28121.701,E2 -28121.701} C_VEL
LIN {X 0,Y 89.587,Z 455.496,A -85,B 0,C 180,E1 -28125.08,E2 -28125.08} C_VEL
LIN {X 0,Y 85.352,Z 457.433,A -85,B 0,C 180,E1 -28128.79,E2 -28128.79} C_VEL
LIN {X 0,Y 81.436,Z 458.937,A -85,B 0,C 180,E1 -28132.828,E2 -28132.828} C_VEL
LIN {X 0,Y 75.088,Z 460.725,A -85,B 0,C 180,E1 -28142.088,E2 -28142.088} C_VEL
LIN {X 0,Y 71.233,Z 461.012,A -85,B 0,C 180,E1 -28152.774,E2 -28152.774} C_VEL
LIN {X 0,Y 69.893,Z 459.688,A -85,B 0,C 180,E1 -28164.219,E2 -28164.219} C_VEL
LIN {X 0,Y 70.022,Z 458.434,A -85,B 0,C 180,E1 -28169.989,E2 -28169.989} C_VEL
LIN {X 0,Y 70.004,Z 455.64,A -85,B 0,C 180,E1 -28178.649,E2 -28178.649} C_VEL
LIN {X 0,Y 71.143,Z 451.778,A -85,B 0,C 180,E1 -28187.226,E2 -28187.226} C_VEL
LIN {X 0,Y 73.658,Z 446.76,A -85,B 0,C 180,E1 -28195.413,E2 -28195.413} C_VEL
LIN {X 0,Y 77.533,Z 440.44,A -85,B 0,C 180,E1 -28202.932,E2 -28202.932} C_VEL
LIN {X 0,Y 81.468,Z 434.116,A -85,B 0,C 180,E1 -28208.504,E2 -28208.504} C_VEL
LIN {X 0,Y 86.583,Z 426.193,A -85,B 0,C 180,E1 -28213.609,E2 -28213.609} C_VEL
LIN {X 0,Y 91.942,Z 416.671,A -85,B 0,C 180,E1 -28218.165,E2 -28218.165} C_VEL
LIN {X 0,Y 96.688,Z 407.407,A -85,B 0,C 180,E1 -28221.369,E2 -28221.369} C_VEL
LIN {X 0,Y 101.108,Z 397.548,A -85,B 0,C 180,E1 -28223.886,E2 -28223.886} C_VEL
LIN {X 0,Y 105.76,Z 385.057,A -85,B 0,C 180,E1 -28226.145,E2 -28226.145} C_VEL
LIN {X 0,Y 108.848,Z 374.136,A -85,B 0,C 180,E1 -28227.578,E2 -28227.578} C_VEL
LIN {X 0,Y 111.399,Z 361.792,A -85,B 0,C 180,E1 -28228.68,E2 -28228.68} C_VEL
LIN {X 0,Y 113.167,Z 346.577,A -85,B 0,C 180,E1 -28229.496,E2 -28229.496} C_VEL
LIN {X 0,Y 115.112,Z 324.267,A -85,B 0,C 180,E1 -28230.513,E2 -28230.513} C_VEL
LIN {X 0,Y 114.98,Z 320.82,A -85,B 0,C 180,E1 -28230.98,E2 -28230.98} C_VEL
LIN {X 0,Y 112.955,Z 313.577,A -85,B 0,C 180,E1 -28233.346,E2 -28233.346} C_VEL
LIN {X 0,Y 111.669,Z 309.938,A -85,B 0,C 180,E1 -28234.861,E2 -28234.861} C_VEL
LIN {X 0,Y 108.495,Z 303.801,A -85,B 0,C 180,E1 -28238.694,E2 -28238.694} C_VEL
LIN {X 0,Y 106.412,Z 300.124,A -85,B 0,C 180,E1 -28241.575,E2 -28241.575} C_VEL
LIN {X 0,Y 104.544,Z 297.013,A -85,B 0,C 180,E1 -28244.543,E2 -28244.543} C_VEL
LIN {X 0,Y 103.167,Z 294.548,A -85,B 0,C 180,E1 -28247.134,E2 -28247.134} C_VEL
LIN {X 0,Y 103.006,Z 294.381,A -85,B 0,C 180,E1 -28247.438,E2 -28247.438} C_VEL
LIN {X 0,Y 101.458,Z 293.274,A -85,B 0,C 180,E1 -28250.587,E2 -28250.587} C_VEL
LIN {X 0,Y 100.093,Z 293.058,A -85,B 0,C 180,E1 -28253.881,E2 -28253.881} C_VEL
LIN {X 0,Y 97.748,Z 294.717,A -85,B 0,C 180,E1 -28265.427,E2 -28265.427} C_VEL
LIN {X 0,Y 98.028,Z 295.756,A -85,B 0,C 180,E1 -28271.198,E2 -28271.198} C_VEL
LIN {X 0,Y 99.406,Z 297.487,A -85,B 0,C 180,E1 -28277.488,E2 -28277.488} C_VEL
LIN {X 0,Y 101.275,Z 300.977,A -85,B 0,C 180,E1 -28282.738,E2 -28282.738} C_VEL
LIN {X 0,Y 102.27,Z 302.661,A -85,B 0,C 180,E1 -28284.864,E2 -28284.864} C_VEL
LIN {X 0,Y 104.284,Z 306.183,A -85,B 0,C 180,E1 -28288.504,E2 -28288.504} C_VEL
LIN {X 0,Y 107.435,Z 312.281,A -85,B 0,C 180,E1 -28293.157,E2 -28293.157} C_VEL
LIN {X 0,Y 110.768,Z 319.786,A -85,B 0,C 180,E1 -28297.309,E2 -28297.309} C_VEL
LIN {X 0,Y 111.341,Z 321.6,A -85,B 0,C 180,E1 -28298.015,E2 -28298.015} C_VEL
LIN {X 0,Y 108.252,Z 352.233,A -85,B 0,C 180,E1 -28299.384,E2 -28299.384} C_VEL
LIN {X 0,Y 105.76,Z 365.689,A -85,B 0,C 180,E1 -28300.499,E2 -28300.499} C_VEL
LIN {X 0,Y 102.419,Z 378.151,A -85,B 0,C 180,E1 -28302.119,E2 -28302.119} C_VEL
LIN {X 0,Y 98.262,Z 389.921,A -85,B 0,C 180,E1 -28304.355,E2 -28304.355} C_VEL
LIN {X 0,Y 93.128,Z 401.296,A -85,B 0,C 180,E1 -28307.235,E2 -28307.235} C_VEL
LIN {X 0,Y 88.161,Z 410.507,A -85,B 0,C 180,E1 -28310.392,E2 -28310.392} C_VEL
LIN {X 0,Y 82.478,Z 419.948,A -85,B 0,C 180,E1 -28314.903,E2 -28314.903} C_VEL
LIN {X 0,Y 76.364,Z 429.036,A -85,B 0,C 180,E1 -28321.122,E2 -28321.122} C_VEL
LIN {X 0,Y 71.082,Z 436.378,A -85,B 0,C 180,E1 -28328.251,E2 -28328.251} C_VEL
LIN {X 0,Y 67.717,Z 441.339,A -85,B 0,C 180,E1 -28334.975,E2 -28334.975} C_VEL
LIN {X 0,Y 64.765,Z 446.172,A -85,B 0,C 180,E1 -28343.783,E2 -28343.783} C_VEL
LIN {X 0,Y 63.276,Z 449.346,A -85,B 0,C 180,E1 -28351.548,E2 -28351.548} C_VEL
LIN {X 0,Y 62.56,Z 452.649,A -85,B 0,C 180,E1 -28362.995,E2 -28362.995} C_VEL
LIN {X 0,Y 63.14,Z 453.95,A -85,B 0,C 180,E1 -28369.518,E2 -28369.518} C_VEL
LIN {X 0,Y 64.466,Z 454.833,A -85,B 0,C 180,E1 -28375.864,E2 -28375.864} C_VEL
LIN {X 0,Y 66.677,Z 455.297,A -85,B 0,C 180,E1 -28382.516,E2 -28382.516} C_VEL
LIN {X 0,Y 72.196,Z 454.992,A -85,B 0,C 180,E1 -28392.964,E2 -28392.964} C_VEL
LIN {X 0,Y 75.934,Z 454.218,A -85,B 0,C 180,E1 -28397.777,E2 -28397.777} C_VEL
LIN {X 0,Y 80.114,Z 453.007,A -85,B 0,C 180,E1 -28402.149,E2 -28402.149} C_VEL
LIN {X 0,Y 87.126,Z 450.388,A -85,B 0,C 180,E1 -28407.892,E2 -28407.892} C_VEL
LIN {X 0,Y 94.872,Z 446.709,A -85,B 0,C 180,E1 -28412.748,E2 -28412.748} C_VEL
LIN {X 0,Y 103.167,Z 441.861,A -85,B 0,C 180,E1 -28416.881,E2 -28416.881} C_VEL
LIN {X 0,Y 111.917,Z 435.691,A -85,B 0,C 180,E1 -28420.386,E2 -28420.386} C_VEL
LIN {X 0,Y 121.155,Z 427.816,A -85,B 0,C 180,E1 -28423.436,E2 -28423.436} C_VEL
LIN {X 0,Y 128.815,Z 419.962,A -85,B 0,C 180,E1 -28425.565,E2 -28425.565} C_VEL
LIN {X 0,Y 136.763,Z 410.144,A -85,B 0,C 180,E1 -28427.521,E2 -28427.521} C_VEL
LIN {X 0,Y 144.026,Z 399.167,A -85,B 0,C 180,E1 -28429.122,E2 -28429.122} C_VEL
LIN {X 0,Y 149.712,Z 388.336,A -85,B 0,C 180,E1 -28430.335,E2 -28430.335} C_VEL
LIN {X 0,Y 154.947,Z 375.65,A -85,B 0,C 180,E1 -28431.252,E2 -28431.252} C_VEL
LIN {X 0,Y 158.763,Z 362.865,A -85,B 0,C 180,E1 -28431.94,E2 -28431.94} C_VEL
LIN {X 0,Y 158.905,Z 362.016,A -85,B 0,C 180,E1 -28432.056,E2 -28432.056} C_VEL
LIN {X 0,Y 157.885,Z 358.088,A -85,B 0,C 180,E1 -28435.692,E2 -28435.692} C_VEL
LIN {X 0,Y 157.279,Z 355.838,A -85,B 0,C 180,E1 -28438.399,E2 -28438.399} C_VEL
LIN {X 0,Y 156.841,Z 353.275,A -85,B 0,C 180,E1 -28442.568,E2 -28442.568} C_VEL
LIN {X 0,Y 156.797,Z 353.389,A -85,B 0,C 180,E1 -28447.404,E2 -28447.404} C_VEL
LIN {X 0,Y 157.682,Z 357.006,A -85,B 0,C 180,E1 -28453.366,E2 -28453.366} C_VEL
LIN {X 0,Y 158.289,Z 360.135,A -85,B 0,C 180,E1 -28455.945,E2 -28455.945} C_VEL
LIN {X 0,Y 158.791,Z 364.241,A -85,B 0,C 180,E1 -28458.406,E2 -28458.406} C_VEL
LIN {X 0,Y 155.364,Z 376.591,A -85,B 0,C 180,E1 -28458.972,E2 -28458.972} C_VEL
LIN {X 0,Y 150.53,Z 388.928,A -85,B 0,C 180,E1 -28459.71,E2 -28459.71} C_VEL
LIN {X 0,Y 144.554,Z 400.554,A -85,B 0,C 180,E1 -28460.625,E2 -28460.625} C_VEL
LIN {X 0,Y 137.314,Z 411.873,A -85,B 0,C 180,E1 -28461.924,E2 -28461.924} C_VEL
LIN {X 0,Y 130.167,Z 420.995,A -85,B 0,C 180,E1 -28463.382,E2 -28463.382} C_VEL
LIN {X 0,Y 122.342,Z 429.362,A -85,B 0,C 180,E1 -28465.206,E2 -28465.206} C_VEL
LIN {X 0,Y 113.309,Z 437.558,A -85,B 0,C 180,E1 -28467.886,E2 -28467.886} C_VEL
LIN {X 0,Y 104.511,Z 444.187,A -85,B 0,C 180,E1 -28470.97,E2 -28470.97} C_VEL
LIN {X 0,Y 94.774,Z 450.281,A -85,B 0,C 180,E1 -28475.336,E2 -28475.336} C_VEL
LIN {X 0,Y 85.493,Z 455.01,A -85,B 0,C 180,E1 -28481.12,E2 -28481.12} C_VEL
LIN {X 0,Y 80.125,Z 457.264,A -85,B 0,C 180,E1 -28485.428,E2 -28485.428} C_VEL
LIN {X 0,Y 72.134,Z 459.766,A -85,B 0,C 180,E1 -28494.218,E2 -28494.218} C_VEL
LIN {X 0,Y 66.329,Z 460.746,A -85,B 0,C 180,E1 -28504.913,E2 -28504.913} C_VEL
LIN {X 0,Y 64.463,Z 460.644,A -85,B 0,C 180,E1 -28510.898,E2 -28510.898} C_VEL
LIN {X 0,Y 62.839,Z 459.259,A -85,B 0,C 180,E1 -28523.567,E2 -28523.567} C_VEL
LIN {X 0,Y 62.926,Z 457.975,A -85,B 0,C 180,E1 -28529.988,E2 -28529.988} C_VEL
LIN {X 0,Y 62.974,Z 455.117,A -85,B 0,C 180,E1 -28539.624,E2 -28539.624} C_VEL
LIN {X 0,Y 64.347,Z 451.187,A -85,B 0,C 180,E1 -28549.113,E2 -28549.113} C_VEL
LIN {X 0,Y 67.294,Z 446.101,A -85,B 0,C 180,E1 -28558.016,E2 -28558.016} C_VEL
LIN {X 0,Y 71.621,Z 439.684,A -85,B 0,C 180,E1 -28566.052,E2 -28566.052} C_VEL
LIN {X 0,Y 77.025,Z 431.793,A -85,B 0,C 180,E1 -28572.963,E2 -28572.963} C_VEL
LIN {X 0,Y 82.642,Z 423.429,A -85,B 0,C 180,E1 -28578.063,E2 -28578.063} C_VEL
LIN {X 0,Y 88.491,Z 413.37,A -85,B 0,C 180,E1 -28582.559,E2 -28582.559} C_VEL
LIN {X 0,Y 94.462,Z 402.106,A -85,B 0,C 180,E1 -28585.841,E2 -28585.841} C_VEL
LIN {X 0,Y 99.154,Z 390.99,A -85,B 0,C 180,E1 -28588.249,E2 -28588.249} C_VEL
LIN {X 0,Y 103.307,Z 378.654,A -85,B 0,C 180,E1 -28590.131,E2 -28590.131} C_VEL
LIN {X 0,Y 106.573,Z 365.562,A -85,B 0,C 180,E1 -28591.399,E2 -28591.399} C_VEL
LIN {X 0,Y 108.626,Z 351.829,A -85,B 0,C 180,E1 -28592.281,E2 -28592.281} C_VEL
LIN {X 0,Y 111.129,Z 325.012,A -85,B 0,C 180,E1 -28593.472,E2 -28593.472} C_VEL
LIN {X 0,Y 110.831,Z 322.483,A -85,B 0,C 180,E1 -28594.028,E2 -28594.028} C_VEL
LIN {X 0,Y 108.84,Z 315.348,A -85,B 0,C 180,E1 -28596.734,E2 -28596.734} C_VEL
LIN {X 0,Y 106.072,Z 309.584,A -85,B 0,C 180,E1 -28600.465,E2 -28600.465} C_VEL
LIN {X 0,Y 103.313,Z 304.28,A -85,B 0,C 180,E1 -28604.927,E2 -28604.927} C_VEL
LIN {X 0,Y 101.375,Z 300.878,A -85,B 0,C 180,E1 -28608.828,E2 -28608.828} C_VEL
LIN {X 0,Y 99.477,Z 297.231,A -85,B 0,C 180,E1 -28614.124,E2 -28614.124} C_VEL
LIN {X 0,Y 97.915,Z 294.674,A -85,B 0,C 180,E1 -28622.44,E2 -28622.44} C_VEL
LIN {X 0,Y 97.748,Z 294.717,A -85,B 0,C 180,E1 -28625.427,E2 -28625.427} C_VEL
LIN {X 0,Y 97.741,Z 295.835,A -85,B 0,C 180,E1 -28628.822,E2 -28628.822} C_VEL
LIN {X 0,Y 97.88,Z 298.179,A -85,B 0,C 180,E1 -28632.027,E2 -28632.027} C_VEL
LIN {X 0,Y 99.329,Z 306.336,A -85,B 0,C 180,E1 -28640.134,E2 -28640.134} C_VEL
LIN {X 0,Y 100.103,Z 307.981,A -85,B 0,C 180,E1 -28642.222,E2 -28642.222} C_VEL
LIN {X 0,Y 102.297,Z 312.353,A -85,B 0,C 180,E1 -28646.88,E2 -28646.88} C_VEL
LIN {X 0,Y 105.026,Z 318.151,A -85,B 0,C 180,E1 -28651.413,E2 -28651.413} C_VEL
LIN {X 0,Y 107.424,Z 324.055,A -85,B 0,C 180,E1 -28654.805,E2 -28654.805} C_VEL
LIN {X 0,Y 106.443,Z 335.03,A -85,B 0,C 180,E1 -28655.359,E2 -28655.359} C_VEL
LIN {X 0,Y 104.268,Z 354.085,A -85,B 0,C 180,E1 -28656.238,E2 -28656.238} C_VEL
LIN {X 0,Y 101.768,Z 366.608,A -85,B 0,C 180,E1 -28657.279,E2 -28657.279} C_VEL
LIN {X 0,Y 98.182,Z 379.125,A -85,B 0,C 180,E1 -28658.9,E2 -28658.9} C_VEL
LIN {X 0,Y 93.455,Z 391.551,A -85,B 0,C 180,E1 -28661.253,E2 -28661.253} C_VEL
LIN {X 0,Y 88.08,Z 402.681,A -85,B 0,C 180,E1 -28664.119,E2 -28664.119} C_VEL
LIN {X 0,Y 82.817,Z 411.716,A -85,B 0,C 180,E1 -28667.26,E2 -28667.26} C_VEL
LIN {X 0,Y 76.773,Z 420.954,A -85,B 0,C 180,E1 -28671.853,E2 -28671.853} C_VEL
LIN {X 0,Y 70.234,Z 429.923,A -85,B 0,C 180,E1 -28678.325,E2 -28678.325} C_VEL
LIN {X 0,Y 64.551,Z 437.166,A -85,B 0,C 180,E1 -28685.918,E2 -28685.918} C_VEL
LIN {X 0,Y 60.884,Z 442.04,A -85,B 0,C 180,E1 -28693.242,E2 -28693.242} C_VEL
LIN {X 0,Y 57.698,Z 446.795,A -85,B 0,C 180,E1 -28703.018,E2 -28703.018} C_VEL
LIN {X 0,Y 56.23,Z 449.594,A -85,B 0,C 180,E1 -28710.738,E2 -28710.738} C_VEL
LIN {X 0,Y 55.538,Z 453.135,A -85,B 0,C 180,E1 -28724.673,E2 -28724.673} C_VEL
LIN {X 0,Y 56.354,Z 454.402,A -85,B 0,C 180,E1 -28731.983,E2 -28731.983} C_VEL
LIN {X 0,Y 60.241,Z 455.618,A -85,B 0,C 180,E1 -28745.248,E2 -28745.248} C_VEL
LIN {X 0,Y 63.398,Z 455.651,A -85,B 0,C 180,E1 -28751.704,E2 -28751.704} C_VEL
LIN {X 0,Y 67.03,Z 455.272,A -85,B 0,C 180,E1 -28757.228,E2 -28757.228} C_VEL
LIN {X 0,Y 75.018,Z 453.44,A -85,B 0,C 180,E1 -28765.798,E2 -28765.798} C_VEL
LIN {X 0,Y 83.471,Z 450.505,A -85,B 0,C 180,E1 -28772.146,E2 -28772.146} C_VEL
LIN {X 0,Y 91.756,Z 446.754,A -85,B 0,C 180,E1 -28776.808,E2 -28776.808} C_VEL
LIN {X 0,Y 100.526,Z 441.828,A -85,B 0,C 180,E1 -28780.71,E2 -28780.71} C_VEL
LIN {X 0,Y 109.682,Z 435.572,A -85,B 0,C 180,E1 -28783.98,E2 -28783.98} C_VEL
LIN {X 0,Y 118.817,Z 427.989,A -85,B 0,C 180,E1 -28786.663,E2 -28786.663} C_VEL
LIN {X 0,Y 127.192,Z 419.57,A -85,B 0,C 180,E1 -28788.75,E2 -28788.75} C_VEL
LIN {X 0,Y 134.553,Z 410.697,A -85,B 0,C 180,E1 -28790.363,E2 -28790.363} C_VEL
LIN {X 0,Y 141.997,Z 399.767,A -85,B 0,C 180,E1 -28791.84,E2 -28791.84} C_VEL
LIN {X 0,Y 147.827,Z 389.039,A -85,B 0,C 180,E1 -28792.947,E2 -28792.947} C_VEL
LIN {X 0,Y 152.981,Z 376.961,A -85,B 0,C 180,E1 -28793.757,E2 -28793.757} C_VEL
LIN {X 0,Y 156.256,Z 366.678,A -85,B 0,C 180,E1 -28794.376,E2 -28794.376} C_VEL
LIN {X 0,Y 155.794,Z 363.766,A -85,B 0,C 180,E1 -28797.414,E2 -28797.414} C_VEL
LIN {X 0,Y 155.584,Z 362.523,A -85,B 0,C 180,E1 -28799.029,E2 -28799.029} C_VEL
LIN {X 0,Y 155.368,Z 360.201,A -85,B 0,C 180,E1 -28803.241,E2 -28803.241} C_VEL
LIN {X 0,Y 155.39,Z 360.353,A -85,B 0,C 180,E1 -28807.144,E2 -28807.144} C_VEL
LIN {X 0,Y 155.971,Z 363.816,A -85,B 0,C 180,E1 -28812.855,E2 -28812.855} C_VEL
LIN {X 0,Y 156.277,Z 367.171,A -85,B 0,C 180,E1 -28815.487,E2 -28815.487} C_VEL
LIN {X 0,Y 156.306,Z 367.981,A -85,B 0,C 180,E1 -28815.985,E2 -28815.985} C_VEL
LIN {X 0,Y 152.588,Z 379.746,A -85,B 0,C 180,E1 -28816.557,E2 -28816.557} C_VEL
LIN {X 0,Y 147.215,Z 392.237,A -85,B 0,C 180,E1 -28817.295,E2 -28817.295} C_VEL
LIN {X 0,Y 140.576,Z 403.976,A -85,B 0,C 180,E1 -28818.214,E2 -28818.214} C_VEL
LIN {X 0,Y 134.032,Z 413.434,A -85,B 0,C 180,E1 -28819.294,E2 -28819.294} C_VEL
LIN {X 0,Y 125.928,Z 423.122,A -85,B 0,C 180,E1 -28820.801,E2 -28820.801} C_VEL
LIN {X 0,Y 117.934,Z 431.084,A -85,B 0,C 180,E1 -28822.526,E2 -28822.526} C_VEL
LIN {X 0,Y 108.631,Z 438.909,A -85,B 0,C 180,E1 -28825.072,E2 -28825.072} C_VEL
LIN {X 0,Y 99.542,Z 445.193,A -85,B 0,C 180,E1 -28828.043,E2 -28828.043} C_VEL
LIN {X 0,Y 90.842,Z 450.222,A -85,B 0,C 180,E1 -28831.671,E2 -28831.671} C_VEL
LIN {X 0,Y 82.7,Z 454.149,A -85,B 0,C 180,E1 -28836.157,E2 -28836.157} C_VEL
LIN {X 0,Y 75.215,Z 457.078,A -85,B 0,C 180,E1 -28841.616,E2 -28841.616} C_VEL
LIN {X 0,Y 66.493,Z 459.511,A -85,B 0,C 180,E1 -28850.631,E2 -28850.631} C_VEL
LIN {X 0,Y 59.935,Z 460.421,A -85,B 0,C 180,E1 -28862.017,E2 -28862.017} C_VEL
LIN {X 0,Y 56.377,Z 459.741,A -85,B 0,C 180,E1 -28875.55,E2 -28875.55} C_VEL
LIN {X 0,Y 55.778,Z 458.828,A -85,B 0,C 180,E1 -28882.749,E2 -28882.749} C_VEL
LIN {X 0,Y 55.822,Z 457.513,A -85,B 0,C 180,E1 -28889.986,E2 -28889.986} C_VEL
LIN {X 0,Y 55.951,Z 454.593,A -85,B 0,C 180,E1 -28900.845,E2 -28900.845} C_VEL
LIN {X 0,Y 57.623,Z 450.595,A -85,B 0,C 180,E1 -28911.446,E2 -28911.446} C_VEL
LIN {X 0,Y 61.834,Z 444.427,A -85,B 0,C 180,E1 -28922.657,E2 -28922.657} C_VEL
LIN {X 0,Y 66.952,Z 437.659,A -85,B 0,C 180,E1 -28930.981,E2 -28930.981} C_VEL
LIN {X 0,Y 71.572,Z 431.434,A -85,B 0,C 180,E1 -28936.47,E2 -28936.47} C_VEL
LIN {X 0,Y 78.053,Z 422.446,A -85,B 0,C 180,E1 -28941.963,E2 -28941.963} C_VEL
LIN {X 0,Y 84.363,Z 412.238,A -85,B 0,C 180,E1 -28946.39,E2 -28946.39} C_VEL
LIN {X 0,Y 90.614,Z 400.718,A -85,B 0,C 180,E1 -28949.612,E2 -28949.612} C_VEL
LIN {X 0,Y 95.591,Z 389.364,A -85,B 0,C 180,E1 -28951.889,E2 -28951.889} C_VEL
LIN {X 0,Y 99.581,Z 377.787,A -85,B 0,C 180,E1 -28953.536,E2 -28953.536} C_VEL
LIN {X 0,Y 102.902,Z 364.719,A -85,B 0,C 180,E1 -28954.723,E2 -28954.723} C_VEL
LIN {X 0,Y 105.009,Z 350.89,A -85,B 0,C 180,E1 -28955.568,E2 -28955.568} C_VEL
LIN {X 0,Y 107.419,Z 326.276,A -85,B 0,C 180,E1 -28956.615,E2 -28956.615} C_VEL
LIN {X 0,Y 105.911,Z 320.301,A -85,B 0,C 180,E1 -28959.009,E2 -28959.009} C_VEL
LIN {X 0,Y 103.569,Z 314.953,A -85,B 0,C 180,E1 -28962.621,E2 -28962.621} C_VEL
LIN {X 0,Y 101.182,Z 310.083,A -85,B 0,C 180,E1 -28967.06,E2 -28967.06} C_VEL
LIN {X 0,Y 99.795,Z 307.306,A -85,B 0,C 180,E1 -28970.302,E2 -28970.302} C_VEL
LIN {X 0,Y 98.085,Z 303.694,A -85,B 0,C 180,E1 -28975.891,E2 -28975.891} C_VEL
LIN {X 0,Y 97.035,Z 301.759,A -85,B 0,C 180,E1 -28982.462,E2 -28982.462} C_VEL
LIN {X 0,Y 96.873,Z 301.967,A -85,B 0,C 180,E1 -28987.118,E2 -28987.118} C_VEL
LIN {X 0,Y 98.198,Z 304.32,A -85,B 0,C 180,E1 -28996.456,E2 -28996.456} C_VEL
LIN {X 0,Y 99.846,Z 307.63,A -85,B 0,C 180,E1 -29001.616,E2 -29001.616} C_VEL
LIN {X 0,Y 100.103,Z 307.981,A -85,B 0,C 180,E1 -29002.222,E2 -29002.222} C_VEL
LIN {X 0,Y 100.829,Z 310.046,A -85,B 0,C 180,E1 -29004.057,E2 -29004.057} C_VEL
LIN {X 0,Y 101.324,Z 313.007,A -85,B 0,C 180,E1 -29005.525,E2 -29005.525} C_VEL
LIN {X 0,Y 102.561,Z 323.338,A -85,B 0,C 180,E1 -29009.267,E2 -29009.267} C_VEL
LIN {X 0,Y 102.817,Z 324.351,A -85,B 0,C 180,E1 -29009.769,E2 -29009.769} C_VEL
LIN {X 0,Y 103.902,Z 327.164,A -85,B 0,C 180,E1 -29011.542,E2 -29011.542} C_VEL
LIN {X 0,Y 101.092,Z 352.908,A -85,B 0,C 180,E1 -29012.67,E2 -29012.67} C_VEL
LIN {X 0,Y 98.286,Z 366.759,A -85,B 0,C 180,E1 -29013.74,E2 -29013.74} C_VEL
LIN {X 0,Y 94.639,Z 379.059,A -85,B 0,C 180,E1 -29015.249,E2 -29015.249} C_VEL
LIN {X 0,Y 89.671,Z 391.567,A -85,B 0,C 180,E1 -29017.503,E2 -29017.503} C_VEL
LIN {X 0,Y 84.009,Z 402.756,A -85,B 0,C 180,E1 -29020.258,E2 -29020.258} C_VEL
LIN {X 0,Y 77.768,Z 412.85,A -85,B 0,C 180,E1 -29023.72,E2 -29023.72} C_VEL
LIN {X 0,Y 71.328,Z 421.94,A -85,B 0,C 180,E1 -29028.33,E2 -29028.33} C_VEL
LIN {X 0,Y 64.284,Z 430.802,A -85,B 0,C 180,E1 -29034.991,E2 -29034.991} C_VEL
LIN {X 0,Y 58.155,Z 437.927,A -85,B 0,C 180,E1 -29043.069,E2 -29043.069} C_VEL
LIN {X 0,Y 54.119,Z 442.735,A -85,B 0,C 180,E1 -29051.072,E2 -29051.072} C_VEL
LIN {X 0,Y 50.639,Z 447.413,A -85,B 0,C 180,E1 -29062.038,E2 -29062.038} C_VEL
LIN {X 0,Y 48.667,Z 451.016,A -85,B 0,C 180,E1 -29074.156,E2 -29074.156} C_VEL
LIN {X 0,Y 48.565,Z 453.618,A -85,B 0,C 180,E1 -29086.838,E2 -29086.838} C_VEL
LIN {X 0,Y 49.708,Z 454.834,A -85,B 0,C 180,E1 -29095.111,E2 -29095.111} C_VEL
LIN {X 0,Y 54.026,Z 455.939,A -85,B 0,C 180,E1 -29108.691,E2 -29108.691} C_VEL
LIN {X 0,Y 58.149,Z 455.971,A -85,B 0,C 180,E1 -29116.496,E2 -29116.496} C_VEL
LIN {X 0,Y 62.295,Z 455.533,A -85,B 0,C 180,E1 -29122.172,E2 -29122.172} C_VEL
LIN {X 0,Y 70.357,Z 453.851,A -85,B 0,C 180,E1 -29130.035,E2 -29130.035} C_VEL
LIN {X 0,Y 80.313,Z 450.624,A -85,B 0,C 180,E1 -29136.766,E2 -29136.766} C_VEL
LIN {X 0,Y 89.129,Z 446.8,A -85,B 0,C 180,E1 -29141.134,E2 -29141.134} C_VEL
LIN {X 0,Y 98.359,Z 441.794,A -85,B 0,C 180,E1 -29144.719,E2 -29144.719} C_VEL
LIN {X 0,Y 107.893,Z 435.445,A -85,B 0,C 180,E1 -29147.716,E2 -29147.716} C_VEL
LIN {X 0,Y 117.683,Z 427.417,A -85,B 0,C 180,E1 -29150.195,E2 -29150.195} C_VEL
LIN {X 0,Y 125.973,Z 419.178,A -85,B 0,C 180,E1 -29152.004,E2 -29152.004} C_VEL
LIN {X 0,Y 133.531,Z 410.163,A -85,B 0,C 180,E1 -29153.429,E2 -29153.429} C_VEL
LIN {X 0,Y 139.95,Z 400.907,A -85,B 0,C 180,E1 -29154.566,E2 -29154.566} C_VEL
LIN {X 0,Y 146.256,Z 389.73,A -85,B 0,C 180,E1 -29155.627,E2 -29155.627} C_VEL
LIN {X 0,Y 151.549,Z 377.635,A -85,B 0,C 180,E1 -29156.364,E2 -29156.364} C_VEL
LIN {X 0,Y 153.497,Z 372.125,A -85,B 0,C 180,E1 -29156.632,E2 -29156.632} C_VEL
LIN {X 0,Y 153.707,Z 371.366,A -85,B 0,C 180,E1 -29156.762,E2 -29156.762} C_VEL
LIN {X 0,Y 153.497,Z 368.387,A -85,B 0,C 180,E1 -29160.984,E2 -29160.984} C_VEL
LIN {X 0,Y 153.573,Z 367.076,A -85,B 0,C 180,E1 -29163.364,E2 -29163.364} C_VEL
LIN {X 0,Y 153.585,Z 367.258,A -85,B 0,C 180,E1 -29166.899,E2 -29166.899} C_VEL
LIN {X 0,Y 153.886,Z 370.02,A -85,B 0,C 180,E1 -29171.86,E2 -29171.86} C_VEL
LIN {X 0,Y 153.909,Z 371.56,A -85,B 0,C 180,E1 -29173.198,E2 -29173.198} C_VEL
LIN {X 0,Y 153.525,Z 373.264,A -85,B 0,C 180,E1 -29173.669,E2 -29173.669} C_VEL
LIN {X 0,Y 149.103,Z 385.048,A -85,B 0,C 180,E1 -29174.191,E2 -29174.191} C_VEL
LIN {X 0,Y 143.579,Z 396.295,A -85,B 0,C 180,E1 -29174.82,E2 -29174.82} C_VEL
LIN {X 0,Y 136.855,Z 407.157,A -85,B 0,C 180,E1 -29175.66,E2 -29175.66} C_VEL
LIN {X 0,Y 130.215,Z 416.016,A -85,B 0,C 180,E1 -29176.662,E2 -29176.662} C_VEL
LIN {X 0,Y 121.949,Z 425.142,A -85,B 0,C 180,E1 -29178.025,E2 -29178.025} C_VEL
LIN {X 0,Y 113.799,Z 432.697,A -85,B 0,C 180,E1 -29179.638,E2 -29179.638} C_VEL
LIN {X 0,Y 104.236,Z 440.126,A -85,B 0,C 180,E1 -29182.01,E2 -29182.01} C_VEL
LIN {X 0,Y 93.337,Z 447.017,A -85,B 0,C 180,E1 -29185.363,E2 -29185.363} C_VEL
LIN {X 0,Y 84.375,Z 451.592,A -85,B 0,C 180,E1 -29188.994,E2 -29188.994} C_VEL
LIN {X 0,Y 75.306,Z 455.343,A -85,B 0,C 180,E1 -29194.052,E2 -29194.052} C_VEL
LIN {X 0,Y 65.69,Z 458.264,A -85,B 0,C 180,E1 -29201.493,E2 -29201.493} C_VEL
LIN {X 0,Y 57.099,Z 459.874,A -85,B 0,C 180,E1 -29212.005,E2 -29212.005} C_VEL
LIN {X 0,Y 51.212,Z 459.899,A -85,B 0,C 180,E1 -29225.675,E2 -29225.675} C_VEL
LIN {X 0,Y 48.75,Z 458.399,A -85,B 0,C 180,E1 -29241.696,E2 -29241.696} C_VEL
LIN {X 0,Y 48.727,Z 457.035,A -85,B 0,C 180,E1 -29249.984,E2 -29249.984} C_VEL
LIN {X 0,Y 48.973,Z 454.061,A -85,B 0,C 180,E1 -29262.414,E2 -29262.414} C_VEL
LIN {X 0,Y 51.036,Z 449.994,A -85,B 0,C 180,E1 -29274.382,E2 -29274.382} C_VEL
LIN {X 0,Y 55.947,Z 443.728,A -85,B 0,C 180,E1 -29286.612,E2 -29286.612} C_VEL
LIN {X 0,Y 61.731,Z 436.878,A -85,B 0,C 180,E1 -29295.338,E2 -29295.338} C_VEL
LIN {X 0,Y 66.35,Z 431.181,A -85,B 0,C 180,E1 -29300.456,E2 -29300.456} C_VEL
LIN {X 0,Y 72.534,Z 423.263,A -85,B 0,C 180,E1 -29305.419,E2 -29305.419} C_VEL
LIN {X 0,Y 79.193,Z 413.298,A -85,B 0,C 180,E1 -29309.884,E2 -29309.884} C_VEL
LIN {X 0,Y 85.039,Z 403.593,A -85,B 0,C 180,E1 -29312.647,E2 -29312.647} C_VEL
LIN {X 0,Y 90.204,Z 393.071,A -85,B 0,C 180,E1 -29314.89,E2 -29314.89} C_VEL
LIN {X 0,Y 94.701,Z 381.497,A -85,B 0,C 180,E1 -29316.657,E2 -29316.657} C_VEL
LIN {X 0,Y 98.553,Z 368.466,A -85,B 0,C 180,E1 -29317.946,E2 -29317.946} C_VEL
LIN {X 0,Y 101.017,Z 355.824,A -85,B 0,C 180,E1 -29318.799,E2 -29318.799} C_VEL
LIN {X 0,Y 103.937,Z 328.605,A -85,B 0,C 180,E1 -29319.924,E2 -29319.924} C_VEL
LIN {X 0,Y 102.979,Z 324.736,A -85,B 0,C 180,E1 -29321.693,E2 -29321.693} C_VEL
LIN {X 0,Y 100.847,Z 319.477,A -85,B 0,C 180,E1 -29325.616,E2 -29325.616} C_VEL
LIN {X 0,Y 98.908,Z 315.131,A -85,B 0,C 180,E1 -29330.057,E2 -29330.057} C_VEL
LIN {X 0,Y 98.116,Z 313.542,A -85,B 0,C 180,E1 -29332.282,E2 -29332.282} C_VEL
LIN {X 0,Y 96.882,Z 310.51,A -85,B 0,C 180,E1 -29337.151,E2 -29337.151} C_VEL
LIN {X 0,Y 96.132,Z 308.854,A -85,B 0,C 180,E1 -29342.717,E2 -29342.717} C_VEL
LIN {X 0,Y 95.998,Z 309.039,A -85,B 0,C 180,E1 -29347.123,E2 -29347.123} C_VEL
LIN {X 0,Y 97.021,Z 311.16,A -85,B 0,C 180,E1 -29355.392,E2 -29355.392} C_VEL
LIN {X 0,Y 98.829,Z 315.14,A -85,B 0,C 180,E1 -29361.509,E2 -29361.509} C_VEL
LIN {X 0,Y 100.329,Z 318.357,A -85,B 0,C 180,E1 -29365.049,E2 -29365.049} C_VEL
LIN {X 0,Y 102.721,Z 324.065,A -85,B 0,C 180,E1 -29369.599,E2 -29369.599} C_VEL
LIN {X 0,Y 102.817,Z 324.351,A -85,B 0,C 180,E1 -29369.769,E2 -29369.769} C_VEL
LIN {X 0,Y 103.045,Z 326.77,A -85,B 0,C 180,E1 -29370.46,E2 -29370.46} C_VEL
LIN {X 0,Y 102.671,Z 330.236,A -85,B 0,C 180,E1 -29370.579,E2 -29370.579} C_VEL
LIN {X 0,Y 101.805,Z 334.037,A -85,B 0,C 180,E1 -29370.147,E2 -29370.147} C_VEL
LIN {X 0,Y 99.613,Z 342.346,A -85,B 0,C 180,E1 -29368.743,E2 -29368.743} C_VEL
LIN {X 0,Y 99.157,Z 345.242,A -85,B 0,C 180,E1 -29368.65,E2 -29368.65} C_VEL
LIN {X 0,Y 97.138,Z 358.563,A -85,B 0,C 180,E1 -29369.318,E2 -29369.318} C_VEL
LIN {X 0,Y 93.95,Z 371.411,A -85,B 0,C 180,E1 -29370.423,E2 -29370.423} C_VEL
LIN {X 0,Y 90.015,Z 382.925,A -85,B 0,C 180,E1 -29371.913,E2 -29371.913} C_VEL
LIN {X 0,Y 84.812,Z 394.665,A -85,B 0,C 180,E1 -29374.063,E2 -29374.063} C_VEL
LIN {X 0,Y 78.92,Z 405.229,A -85,B 0,C 180,E1 -29376.753,E2 -29376.753} C_VEL
LIN {X 0,Y 73.049,Z 413.951,A -85,B 0,C 180,E1 -29379.698,E2 -29379.698} C_VEL
LIN {X 0,Y 66.201,Z 422.911,A -85,B 0,C 180,E1 -29384.249,E2 -29384.249} C_VEL
LIN {X 0,Y 58.604,Z 431.665,A -85,B 0,C 180,E1 -29391.001,E2 -29391.001} C_VEL
LIN {X 0,Y 51.942,Z 438.654,A -85,B 0,C 180,E1 -29399.53,E2 -29399.53} C_VEL
LIN {X 0,Y 45.896,Z 445.061,A -85,B 0,C 180,E1 -29412.185,E2 -29412.185} C_VEL
LIN {X 0,Y 42.489,Z 449.566,A -85,B 0,C 180,E1 -29426.313,E2 -29426.313} C_VEL
LIN {X 0,Y 41.255,Z 452.491,A -85,B 0,C 180,E1 -29439.826,E2 -29439.826} C_VEL
LIN {X 0,Y 41.701,Z 454.097,A -85,B 0,C 180,E1 -29449.716,E2 -29449.716} C_VEL
LIN {X 0,Y 43.261,Z 455.249,A -85,B 0,C 180,E1 -29459.184,E2 -29459.184} C_VEL
LIN {X 0,Y 47.996,Z 456.259,A -85,B 0,C 180,E1 -29472.932,E2 -29472.932} C_VEL
LIN {X 0,Y 53.381,Z 456.286,A -85,B 0,C 180,E1 -29482.196,E2 -29482.196} C_VEL
LIN {X 0,Y 58.098,Z 455.788,A -85,B 0,C 180,E1 -29487.878,E2 -29487.878} C_VEL
LIN {X 0,Y 66.134,Z 454.262,A -85,B 0,C 180,E1 -29494.844,E2 -29494.844} C_VEL
LIN {X 0,Y 77.717,Z 450.744,A -85,B 0,C 180,E1 -29501.733,E2 -29501.733} C_VEL
LIN {X 0,Y 88.529,Z 446.139,A -85,B 0,C 180,E1 -29506.222,E2 -29506.222} C_VEL
LIN {X 0,Y 99.963,Z 439.746,A -85,B 0,C 180,E1 -29509.839,E2 -29509.839} C_VEL
LIN {X 0,Y 109.31,Z 433.244,A -85,B 0,C 180,E1 -29512.198,E2 -29512.198} C_VEL
LIN {X 0,Y 118.356,Z 425.635,A -85,B 0,C 180,E1 -29514.062,E2 -29514.062} C_VEL
LIN {X 0,Y 126.877,Z 416.909,A -85,B 0,C 180,E1 -29515.61,E2 -29515.61} C_VEL
LIN {X 0,Y 134.983,Z 406.786,A -85,B 0,C 180,E1 -29516.852,E2 -29516.852} C_VEL
LIN {X 0,Y 142.403,Z 395.237,A -85,B 0,C 180,E1 -29518.003,E2 -29518.003} C_VEL
LIN {X 0,Y 147.625,Z 385.013,A -85,B 0,C 180,E1 -29518.69,E2 -29518.69} C_VEL
LIN {X 0,Y 150.706,Z 377.6,A -85,B 0,C 180,E1 -29519.041,E2 -29519.041} C_VEL
LIN {X 0,Y 151.117,Z 376.361,A -85,B 0,C 180,E1 -29519.334,E2 -29519.334} C_VEL
LIN {X 0,Y 151.322,Z 374.304,A -85,B 0,C 180,E1 -29522.662,E2 -29522.662} C_VEL
LIN {X 0,Y 151.415,Z 373.772,A -85,B 0,C 180,E1 -29525.326,E2 -29525.326} C_VEL
LIN {X 0,Y 151.479,Z 376.385,A -85,B 0,C 180,E1 -29531.03,E2 -29531.03} C_VEL
LIN {X 0,Y 150.474,Z 379.128,A -85,B 0,C 180,E1 -29531.242,E2 -29531.242} C_VEL
LIN {X 0,Y 145.595,Z 390.271,A -85,B 0,C 180,E1 -29531.728,E2 -29531.728} C_VEL
LIN {X 0,Y 139.375,Z 401.394,A -85,B 0,C 180,E1 -29532.315,E2 -29532.315} C_VEL
LIN {X 0,Y 131.725,Z 412.274,A -85,B 0,C 180,E1 -29533.168,E2 -29533.168} C_VEL
LIN {X 0,Y 123.288,Z 422.046,A -85,B 0,C 180,E1 -29534.282,E2 -29534.282} C_VEL
LIN {X 0,Y 114.908,Z 430.077,A -85,B 0,C 180,E1 -29535.567,E2 -29535.567} C_VEL
LIN {X 0,Y 105.049,Z 437.976,A -85,B 0,C 180,E1 -29537.563,E2 -29537.563} C_VEL
LIN {X 0,Y 96.925,Z 443.344,A -85,B 0,C 180,E1 -29539.495,E2 -29539.495} C_VEL
LIN {X 0,Y 87.369,Z 448.626,A -85,B 0,C 180,E1 -29542.312,E2 -29542.312} C_VEL
LIN {X 0,Y 78.135,Z 452.762,A -85,B 0,C 180,E1 -29545.901,E2 -29545.901} C_VEL
LIN {X 0,Y 70.696,Z 455.458,A -85,B 0,C 180,E1 -29549.805,E2 -29549.805} C_VEL
LIN {X 0,Y 61.207,Z 458.043,A -85,B 0,C 180,E1 -29556.496,E2 -29556.496} C_VEL
LIN {X 0,Y 51.684,Z 459.579,A -85,B 0,C 180,E1 -29567.149,E2 -29567.149} C_VEL
LIN {X 0,Y 44.8,Z 459.523,A -85,B 0,C 180,E1 -29581.909,E2 -29581.909} C_VEL
LIN {X 0,Y 41.716,Z 457.963,A -85,B 0,C 180,E1 -29600.283,E2 -29600.283} C_VEL
LIN {X 0,Y 41.621,Z 456.54,A -85,B 0,C 180,E1 -29609.982,E2 -29609.982} C_VEL
LIN {X 0,Y 42.033,Z 453.502,A -85,B 0,C 180,E1 -29624.505,E2 -29624.505} C_VEL
LIN {X 0,Y 44.627,Z 449.363,A -85,B 0,C 180,E1 -29638.171,E2 -29638.171} C_VEL
LIN {X 0,Y 50.389,Z 443.015,A -85,B 0,C 180,E1 -29651.466,E2 -29651.466} C_VEL
LIN {X 0,Y 56.916,Z 436.075,A -85,B 0,C 180,E1 -29660.483,E2 -29660.483} C_VEL
LIN {X 0,Y 61.861,Z 430.499,A -85,B 0,C 180,E1 -29665.387,E2 -29665.387} C_VEL
LIN {X 0,Y 68.732,Z 422.25,A -85,B 0,C 180,E1 -29670.328,E2 -29670.328} C_VEL
LIN {X 0,Y 75.881,Z 412.155,A -85,B 0,C 180,E1 -29674.525,E2 -29674.525} C_VEL
LIN {X 0,Y 82.749,Z 400.788,A -85,B 0,C 180,E1 -29677.425,E2 -29677.425} C_VEL
LIN {X 0,Y 88.177,Z 389.603,A -85,B 0,C 180,E1 -29679.434,E2 -29679.434} C_VEL
LIN {X 0,Y 92.901,Z 377.136,A -85,B 0,C 180,E1 -29680.979,E2 -29680.979} C_VEL
LIN {X 0,Y 96.526,Z 363.742,A -85,B 0,C 180,E1 -29682.009,E2 -29682.009} C_VEL
LIN {X 0,Y 98.692,Z 350.55,A -85,B 0,C 180,E1 -29682.719,E2 -29682.719} C_VEL
LIN {X 0,Y 100.786,Z 331.045,A -85,B 0,C 180,E1 -29683.459,E2 -29683.459} C_VEL
LIN {X 0,Y 99.655,Z 327.444,A -85,B 0,C 180,E1 -29685.84,E2 -29685.84} C_VEL
LIN {X 0,Y 97.687,Z 322.344,A -85,B 0,C 180,E1 -29690.685,E2 -29690.685} C_VEL
LIN {X 0,Y 96.729,Z 320.044,A -85,B 0,C 180,E1 -29693.744,E2 -29693.744} C_VEL
LIN {X 0,Y 95.835,Z 317.428,A -85,B 0,C 180,E1 -29697.899,E2 -29697.899} C_VEL
LIN {X 0,Y 95.173,Z 315.779,A -85,B 0,C 180,E1 -29704.235,E2 -29704.235} C_VEL
LIN {X 0,Y 95.239,Z 316.749,A -85,B 0,C 180,E1 -29709.827,E2 -29709.827} C_VEL
LIN {X 0,Y 95.911,Z 318.089,A -85,B 0,C 180,E1 -29714.479,E2 -29714.479} C_VEL
LIN {X 0,Y 97.368,Z 321.686,A -85,B 0,C 180,E1 -29720.135,E2 -29720.135} C_VEL
LIN {X 0,Y 98.893,Z 325.403,A -85,B 0,C 180,E1 -29724.169,E2 -29724.169} C_VEL
LIN {X 0,Y 100.697,Z 330.55,A -85,B 0,C 180,E1 -29728.057,E2 -29728.057} C_VEL
LIN {X 0,Y 99.157,Z 345.242,A -85,B 0,C 180,E1 -29728.65,E2 -29728.65} C_VEL
LIN {X 0,Y 98.419,Z 349.164,A -85,B 0,C 180,E1 -29728.418,E2 -29728.418} C_VEL
LIN {X 0,Y 94.196,Z 361.282,A -85,B 0,C 180,E1 -29725.839,E2 -29725.839} C_VEL
LIN {X 0,Y 93.076,Z 365.085,A -85,B 0,C 180,E1 -29725.794,E2 -29725.794} C_VEL
LIN {X 0,Y 89.351,Z 377.367,A -85,B 0,C 180,E1 -29726.989,E2 -29726.989} C_VEL
LIN {X 0,Y 84.181,Z 389.987,A -85,B 0,C 180,E1 -29728.793,E2 -29728.793} C_VEL
LIN {X 0,Y 77.946,Z 401.584,A -85,B 0,C 180,E1 -29731.095,E2 -29731.095} C_VEL
LIN {X 0,Y 71.754,Z 410.975,A -85,B 0,C 180,E1 -29733.667,E2 -29733.667} C_VEL
LIN {X 0,Y 64.343,Z 420.574,A -85,B 0,C 180,E1 -29737.664,E2 -29737.664} C_VEL
LIN {X 0,Y 57.315,Z 428.435,A -85,B 0,C 180,E1 -29742.657,E2 -29742.657} C_VEL
LIN {X 0,Y 49.445,Z 436.129,A -85,B 0,C 180,E1 -29750.262,E2 -29750.262} C_VEL
LIN {X 0,Y 42.824,Z 442.291,A -85,B 0,C 180,E1 -29760.529,E2 -29760.529} C_VEL
LIN {X 0,Y 37.751,Z 447.202,A -85,B 0,C 180,E1 -29773.807,E2 -29773.807} C_VEL
LIN {X 0,Y 34.752,Z 451.015,A -85,B 0,C 180,E1 -29790.022,E2 -29790.022} C_VEL
LIN {X 0,Y 34.16,Z 453.005,A -85,B 0,C 180,E1 -29801.894,E2 -29801.894} C_VEL
LIN {X 0,Y 34.975,Z 454.564,A -85,B 0,C 180,E1 -29813.717,E2 -29813.717} C_VEL
LIN {X 0,Y 40.355,Z 456.368,A -85,B 0,C 180,E1 -29834.177,E2 -29834.177} C_VEL
LIN {X 0,Y 44.457,Z 456.686,A -85,B 0,C 180,E1 -29842.246,E2 -29842.246} C_VEL
LIN {X 0,Y 49.234,Z 456.582,A -85,B 0,C 180,E1 -29848.945,E2 -29848.945} C_VEL
LIN {X 0,Y 60.296,Z 455.102,A -85,B 0,C 180,E1 -29858.842,E2 -29858.842} C_VEL
LIN {X 0,Y 66.309,Z 453.756,A -85,B 0,C 180,E1 -29862.555,E2 -29862.555} C_VEL
LIN {X 0,Y 75.749,Z 450.863,A -85,B 0,C 180,E1 -29866.974,E2 -29866.974} C_VEL
LIN {X 0,Y 86.107,Z 446.621,A -85,B 0,C 180,E1 -29870.605,E2 -29870.605} C_VEL
LIN {X 0,Y 97.242,Z 440.689,A -85,B 0,C 180,E1 -29873.614,E2 -29873.614} C_VEL
LIN {X 0,Y 108.108,Z 433.408,A -85,B 0,C 180,E1 -29875.916,E2 -29875.916} C_VEL
LIN {X 0,Y 117.826,Z 425.325,A -85,B 0,C 180,E1 -29877.578,E2 -29877.578} C_VEL
LIN {X 0,Y 126.528,Z 416.449,A -85,B 0,C 180,E1 -29878.899,E2 -29878.899} C_VEL
LIN {X 0,Y 135.211,Z 405.575,A -85,B 0,C 180,E1 -29880,E2 -29880} C_VEL
LIN {X 0,Y 141.99,Z 394.935,A -85,B 0,C 180,E1 -29880.887,E2 -29880.887} C_VEL
LIN {X 0,Y 146.865,Z 385.493,A -85,B 0,C 180,E1 -29881.431,E2 -29881.431} C_VEL
LIN {X 0,Y 148.544,Z 381.649,A -85,B 0,C 180,E1 -29881.661,E2 -29881.661} C_VEL
LIN {X 0,Y 148.704,Z 381.042,A -85,B 0,C 180,E1 -29882.709,E2 -29882.709} C_VEL
LIN {X 0,Y 148.882,Z 380.51,A -85,B 0,C 180,E1 -29885.417,E2 -29885.417} C_VEL
LIN {X 0,Y 148.707,Z 381.794,A -85,B 0,C 180,E1 -29888.492,E2 -29888.492} C_VEL
LIN {X 0,Y 147.907,Z 383.695,A -85,B 0,C 180,E1 -29888.71,E2 -29888.71} C_VEL
LIN {X 0,Y 142.355,Z 394.891,A -85,B 0,C 180,E1 -29889.11,E2 -29889.11} C_VEL
LIN {X 0,Y 135.459,Z 405.929,A -85,B 0,C 180,E1 -29889.676,E2 -29889.676} C_VEL
LIN {X 0,Y 128.598,Z 414.883,A -85,B 0,C 180,E1 -29890.351,E2 -29890.351} C_VEL
LIN {X 0,Y 120.037,Z 424.099,A -85,B 0,C 180,E1 -29891.275,E2 -29891.275} C_VEL
LIN {X 0,Y 111.534,Z 431.718,A -85,B 0,C 180,E1 -29892.388,E2 -29892.388} C_VEL
LIN {X 0,Y 101.451,Z 439.203,A -85,B 0,C 180,E1 -29894.097,E2 -29894.097} C_VEL
LIN {X 0,Y 91.486,Z 445.244,A -85,B 0,C 180,E1 -29896.197,E2 -29896.197} C_VEL
LIN {X 0,Y 81.687,Z 450.053,A -85,B 0,C 180,E1 -29898.834,E2 -29898.834} C_VEL
LIN {X 0,Y 72.172,Z 453.772,A -85,B 0,C 180,E1 -29902.303,E2 -29902.303} C_VEL
LIN {X 0,Y 63.063,Z 456.508,A -85,B 0,C 180,E1 -29906.916,E2 -29906.916} C_VEL
LIN {X 0,Y 51.766,Z 458.754,A -85,B 0,C 180,E1 -29915.436,E2 -29915.436} C_VEL
LIN {X 0,Y 42.241,Z 459.392,A -85,B 0,C 180,E1 -29928.259,E2 -29928.259} C_VEL
LIN {X 0,Y 36.1,Z 458.531,A -85,B 0,C 180,E1 -29947.065,E2 -29947.065} C_VEL
LIN {X 0,Y 34.722,Z 457.512,A -85,B 0,C 180,E1 -29958.301,E2 -29958.301} C_VEL
LIN {X 0,Y 34.514,Z 456.042,A -85,B 0,C 180,E1 -29969.978,E2 -29969.978} C_VEL
LIN {X 0,Y 35.18,Z 452.936,A -85,B 0,C 180,E1 -29987.413,E2 -29987.413} C_VEL
LIN {X 0,Y 38.469,Z 448.724,A -85,B 0,C 180,E1 -30003.208,E2 -30003.208} C_VEL
LIN {X 0,Y 45.263,Z 442.297,A -85,B 0,C 180,E1 -30017.491,E2 -30017.491} C_VEL
LIN {X 0,Y 52.48,Z 435.41,A -85,B 0,C 180,E1 -30026.387,E2 -30026.387} C_VEL
LIN {X 0,Y 57.985,Z 429.735,A -85,B 0,C 180,E1 -30031.087,E2 -30031.087} C_VEL
LIN {X 0,Y 65.475,Z 421.233,A -85,B 0,C 180,E1 -30035.795,E2 -30035.795} C_VEL
LIN {X 0,Y 72.31,Z 412.087,A -85,B 0,C 180,E1 -30039.26,E2 -30039.26} C_VEL
LIN {X 0,Y 79.478,Z 400.804,A -85,B 0,C 180,E1 -30041.866,E2 -30041.866} C_VEL
LIN {X 0,Y 85.116,Z 389.7,A -85,B 0,C 180,E1 -30043.662,E2 -30043.662} C_VEL
LIN {X 0,Y 90.034,Z 377.289,A -85,B 0,C 180,E1 -30045.038,E2 -30045.038} C_VEL
LIN {X 0,Y 93.737,Z 364.253,A -85,B 0,C 180,E1 -30045.953,E2 -30045.953} C_VEL
LIN {X 0,Y 95.979,Z 351.738,A -85,B 0,C 180,E1 -30046.555,E2 -30046.555} C_VEL
LIN {X 0,Y 97.987,Z 334.212,A -85,B 0,C 180,E1 -30047.135,E2 -30047.135} C_VEL
LIN {X 0,Y 96.348,Z 329.176,A -85,B 0,C 180,E1 -30051.744,E2 -30051.744} C_VEL
LIN {X 0,Y 95.467,Z 326.72,A -85,B 0,C 180,E1 -30054.985,E2 -30054.985} C_VEL
LIN {X 0,Y 94.674,Z 324.139,A -85,B 0,C 180,E1 -30059.469,E2 -30059.469} C_VEL
LIN {X 0,Y 94.297,Z 322.84,A -85,B 0,C 180,E1 -30064.275,E2 -30064.275} C_VEL
LIN {X 0,Y 94.315,Z 323.722,A -85,B 0,C 180,E1 -30069.247,E2 -30069.247} C_VEL
LIN {X 0,Y 94.803,Z 324.928,A -85,B 0,C 180,E1 -30073.387,E2 -30073.387} C_VEL
LIN {X 0,Y 96.039,Z 328.493,A -85,B 0,C 180,E1 -30079.001,E2 -30079.001} C_VEL
LIN {X 0,Y 97.211,Z 331.841,A -85,B 0,C 180,E1 -30082.588,E2 -30082.588} C_VEL
LIN {X 0,Y 97.878,Z 333.925,A -85,B 0,C 180,E1 -30084.337,E2 -30084.337} C_VEL
LIN {X 0,Y 95.324,Z 354.565,A -85,B 0,C 180,E1 -30085.137,E2 -30085.137} C_VEL
LIN {X 0,Y 93.076,Z 365.085,A -85,B 0,C 180,E1 -30085.794,E2 -30085.794} C_VEL
LIN {X 0,Y 91.334,Z 370.812,A -85,B 0,C 180,E1 -30085.988,E2 -30085.988} C_VEL
LIN {X 0,Y 87.339,Z 379.854,A -85,B 0,C 180,E1 -30085.219,E2 -30085.219} C_VEL
LIN {X 0,Y 82.713,Z 388.528,A -85,B 0,C 180,E1 -30084.432,E2 -30084.432} C_VEL
LIN {X 0,Y 79.949,Z 393.647,A -85,B 0,C 180,E1 -30084.739,E2 -30084.739} C_VEL
LIN {X 0,Y 73.755,Z 404.208,A -85,B 0,C 180,E1 -30086.739,E2 -30086.739} C_VEL
LIN {X 0,Y 66.492,Z 414.199,A -85,B 0,C 180,E1 -30089.342,E2 -30089.342} C_VEL
LIN {X 0,Y 58.753,Z 423.223,A -85,B 0,C 180,E1 -30093.172,E2 -30093.172} C_VEL
LIN {X 0,Y 49.834,Z 432.039,A -85,B 0,C 180,E1 -30099.166,E2 -30099.166} C_VEL
LIN {X 0,Y 41.633,Z 439.095,A -85,B 0,C 180,E1 -30107.558,E2 -30107.558} C_VEL
LIN {X 0,Y 34.607,Z 444.733,A -85,B 0,C 180,E1 -30119.518,E2 -30119.518} C_VEL
LIN {X 0,Y 29.543,Z 449.182,A -85,B 0,C 180,E1 -30136.266,E2 -30136.266} C_VEL
LIN {X 0,Y 27.547,Z 451.561,A -85,B 0,C 180,E1 -30150.027,E2 -30150.027} C_VEL
LIN {X 0,Y 27.121,Z 453.519,A -85,B 0,C 180,E1 -30165.046,E2 -30165.046} C_VEL
LIN {X 0,Y 28.479,Z 455.014,A -85,B 0,C 180,E1 -30179.602,E2 -30179.602} C_VEL
LIN {X 0,Y 31.398,Z 456.079,A -85,B 0,C 180,E1 -30192.21,E2 -30192.21} C_VEL
LIN {X 0,Y 37.061,Z 456.897,A -85,B 0,C 180,E1 -30205.324,E2 -30205.324} C_VEL
LIN {X 0,Y 45.896,Z 456.869,A -85,B 0,C 180,E1 -30216.775,E2 -30216.775} C_VEL
LIN {X 0,Y 58.06,Z 455.324,A -85,B 0,C 180,E1 -30225.583,E2 -30225.583} C_VEL
LIN {X 0,Y 64.495,Z 453.924,A -85,B 0,C 180,E1 -30228.766,E2 -30228.766} C_VEL
LIN {X 0,Y 74.444,Z 450.965,A -85,B 0,C 180,E1 -30232.457,E2 -30232.457} C_VEL
LIN {X 0,Y 84.625,Z 446.911,A -85,B 0,C 180,E1 -30235.304,E2 -30235.304} C_VEL
LIN {X 0,Y 96.703,Z 440.614,A -85,B 0,C 180,E1 -30237.908,E2 -30237.908} C_VEL
LIN {X 0,Y 105.428,Z 434.953,A -85,B 0,C 180,E1 -30239.412,E2 -30239.412} C_VEL
LIN {X 0,Y 115.978,Z 426.607,A -85,B 0,C 180,E1 -30240.894,E2 -30240.894} C_VEL
LIN {X 0,Y 124.823,Z 417.975,A -85,B 0,C 180,E1 -30241.986,E2 -30241.986} C_VEL
LIN {X 0,Y 132.813,Z 408.438,A -85,B 0,C 180,E1 -30242.807,E2 -30242.807} C_VEL
LIN {X 0,Y 139.955,Z 397.959,A -85,B 0,C 180,E1 -30243.59,E2 -30243.59} C_VEL
LIN {X 0,Y 145.275,Z 388.329,A -85,B 0,C 180,E1 -30244.102,E2 -30244.102} C_VEL
LIN {X 0,Y 145.834,Z 387.202,A -85,B 0,C 180,E1 -30244.286,E2 -30244.286} C_VEL
LIN {X 0,Y 145.928,Z 387.096,A -85,B 0,C 180,E1 -30245.527,E2 -30245.527} C_VEL
LIN {X 0,Y 145.282,Z 388.481,A -85,B 0,C 180,E1 -30246.091,E2 -30246.091} C_VEL
LIN {X 0,Y 138.8,Z 400.064,A -85,B 0,C 180,E1 -30246.439,E2 -30246.439} C_VEL
LIN {X 0,Y 130.971,Z 411.113,A -85,B 0,C 180,E1 -30246.913,E2 -30246.913} C_VEL
LIN {X 0,Y 122.314,Z 420.965,A -85,B 0,C 180,E1 -30247.619,E2 -30247.619} C_VEL
LIN {X 0,Y 113.661,Z 429.068,A -85,B 0,C 180,E1 -30248.37,E2 -30248.37} C_VEL
LIN {X 0,Y 103.375,Z 437.033,A -85,B 0,C 180,E1 -30249.661,E2 -30249.661} C_VEL
LIN {X 0,Y 93.156,Z 443.44,A -85,B 0,C 180,E1 -30251.244,E2 -30251.244} C_VEL
LIN {X 0,Y 83.022,Z 448.559,A -85,B 0,C 180,E1 -30253.205,E2 -30253.205} C_VEL
LIN {X 0,Y 73.047,Z 452.563,A -85,B 0,C 180,E1 -30255.803,E2 -30255.803} C_VEL
LIN {X 0,Y 60.173,Z 456.318,A -85,B 0,C 180,E1 -30260.853,E2 -30260.853} C_VEL
LIN {X 0,Y 47.983,Z 458.486,A -85,B 0,C 180,E1 -30268.478,E2 -30268.478} C_VEL
LIN {X 0,Y 37.224,Z 459.048,A -85,B 0,C 180,E1 -30280.932,E2 -30280.932} C_VEL
LIN {X 0,Y 29.66,Z 458.124,A -85,B 0,C 180,E1 -30301.686,E2 -30301.686} C_VEL
LIN {X 0,Y 27.807,Z 457.047,A -85,B 0,C 180,E1 -30315.333,E2 -30315.333} C_VEL
LIN {X 0,Y 27.402,Z 455.544,A -85,B 0,C 180,E1 -30329.972,E2 -30329.972} C_VEL
LIN {X 0,Y 28.445,Z 452.369,A -85,B 0,C 180,E1 -30351.722,E2 -30351.722} C_VEL
LIN {X 0,Y 32.723,Z 448.085,A -85,B 0,C 180,E1 -30370.079,E2 -30370.079} C_VEL
LIN {X 0,Y 40.771,Z 441.581,A -85,B 0,C 180,E1 -30384.924,E2 -30384.924} C_VEL
LIN {X 0,Y 49.454,Z 433.984,A -85,B 0,C 180,E1 -30394.002,E2 -30394.002} C_VEL
LIN {X 0,Y 58.163,Z 425.485,A -85,B 0,C 180,E1 -30399.412,E2 -30399.412} C_VEL
LIN {X 0,Y 66.046,Z 416.284,A -85,B 0,C 180,E1 -30403.215,E2 -30403.215} C_VEL
LIN {X 0,Y 73.404,Z 406.135,A -85,B 0,C 180,E1 -30405.726,E2 -30405.726} C_VEL
LIN {X 0,Y 80.053,Z 394.842,A -85,B 0,C 180,E1 -30407.533,E2 -30407.533} C_VEL
LIN {X 0,Y 85.486,Z 383.118,A -85,B 0,C 180,E1 -30408.859,E2 -30408.859} C_VEL
LIN {X 0,Y 90.044,Z 369.95,A -85,B 0,C 180,E1 -30409.817,E2 -30409.817} C_VEL
LIN {X 0,Y 93.085,Z 356.784,A -85,B 0,C 180,E1 -30410.467,E2 -30410.467} C_VEL
LIN {X 0,Y 95.511,Z 337.894,A -85,B 0,C 180,E1 -30411.099,E2 -30411.099} C_VEL
LIN {X 0,Y 94.42,Z 333.864,A -85,B 0,C 180,E1 -30415.464,E2 -30415.464} C_VEL
LIN {X 0,Y 93.713,Z 331.12,A -85,B 0,C 180,E1 -30420,E2 -30420} C_VEL
LIN {X 0,Y 93.421,Z 329.904,A -85,B 0,C 180,E1 -30424.315,E2 -30424.315} C_VEL
LIN {X 0,Y 93.49,Z 331.02,A -85,B 0,C 180,E1 -30430.013,E2 -30430.013} C_VEL
LIN {X 0,Y 93.797,Z 332.03,A -85,B 0,C 180,E1 -30432.801,E2 -30432.801} C_VEL
LIN {X 0,Y 94.684,Z 335.046,A -85,B 0,C 180,E1 -30437.551,E2 -30437.551} C_VEL
LIN {X 0,Y 95.448,Z 337.69,A -85,B 0,C 180,E1 -30440.423,E2 -30440.423} C_VEL
LIN {X 0,Y 92.96,Z 356.23,A -85,B 0,C 180,E1 -30441.089,E2 -30441.089} C_VEL
LIN {X 0,Y 89.791,Z 369.381,A -85,B 0,C 180,E1 -30441.88,E2 -30441.88} C_VEL
LIN {X 0,Y 85.721,Z 381.111,A -85,B 0,C 180,E1 -30443.016,E2 -30443.016} C_VEL
LIN {X 0,Y 79.949,Z 393.647,A -85,B 0,C 180,E1 -30444.739,E2 -30444.739} C_VEL
LIN {X 0,Y 76.967,Z 398.724,A -85,B 0,C 180,E1 -30445.126,E2 -30445.126} C_VEL
LIN {X 0,Y 71.039,Z 406.653,A -85,B 0,C 180,E1 -30444.528,E2 -30444.528} C_VEL
LIN {X 0,Y 64.523,Z 414.116,A -85,B 0,C 180,E1 -30443.998,E2 -30443.998} C_VEL
LIN {X 0,Y 60.605,Z 418.461,A -85,B 0,C 180,E1 -30444.75,E2 -30444.75} C_VEL
LIN {X 0,Y 52.01,Z 427.29,A -85,B 0,C 180,E1 -30448.599,E2 -30448.599} C_VEL
LIN {X 0,Y 42.592,Z 435.366,A -85,B 0,C 180,E1 -30454.447,E2 -30454.447} C_VEL
LIN {X 0,Y 33.904,Z 441.839,A -85,B 0,C 180,E1 -30463.527,E2 -30463.527} C_VEL
LIN {X 0,Y 26.393,Z 446.99,A -85,B 0,C 180,E1 -30477.859,E2 -30477.859} C_VEL
LIN {X 0,Y 21.487,Z 450.798,A -85,B 0,C 180,E1 -30498.897,E2 -30498.897} C_VEL
LIN {X 0,Y 20.239,Z 454.022,A -85,B 0,C 180,E1 -30530.357,E2 -30530.357} C_VEL
LIN {X 0,Y 22.458,Z 455.462,A -85,B 0,C 180,E1 -30548.786,E2 -30548.786} C_VEL
LIN {X 0,Y 26.472,Z 456.495,A -85,B 0,C 180,E1 -30562.835,E2 -30562.835} C_VEL
LIN {X 0,Y 32.562,Z 457.216,A -85,B 0,C 180,E1 -30574.425,E2 -30574.425} C_VEL
LIN {X 0,Y 43.537,Z 457.156,A -85,B 0,C 180,E1 -30585.643,E2 -30585.643} C_VEL
LIN {X 0,Y 56.68,Z 455.547,A -85,B 0,C 180,E1 -30592.786,E2 -30592.786} C_VEL
LIN {X 0,Y 63.478,Z 454.078,A -85,B 0,C 180,E1 -30595.241,E2 -30595.241} C_VEL
LIN {X 0,Y 73.841,Z 451.049,A -85,B 0,C 180,E1 -30598.097,E2 -30598.097} C_VEL
LIN {X 0,Y 84.342,Z 446.918,A -85,B 0,C 180,E1 -30600.261,E2 -30600.261} C_VEL
LIN {X 0,Y 94.939,Z 441.557,A -85,B 0,C 180,E1 -30601.984,E2 -30601.984} C_VEL
LIN {X 0,Y 105.604,Z 434.787,A -85,B 0,C 180,E1 -30603.355,E2 -30603.355} C_VEL
LIN {X 0,Y 112.743,Z 429.352,A -85,B 0,C 180,E1 -30604.132,E2 -30604.132} C_VEL
LIN {X 0,Y 112.847,Z 429.306,A -85,B 0,C 180,E1 -30604.809,E2 -30604.809} C_VEL
LIN {X 0,Y 102.423,Z 437.158,A -85,B 0,C 180,E1 -30605.74,E2 -30605.74} C_VEL
LIN {X 0,Y 92.035,Z 443.458,A -85,B 0,C 180,E1 -30606.902,E2 -30606.902} C_VEL
LIN {X 0,Y 81.691,Z 448.502,A -85,B 0,C 180,E1 -30608.338,E2 -30608.338} C_VEL
LIN {X 0,Y 71.437,Z 452.439,A -85,B 0,C 180,E1 -30610.298,E2 -30610.298} C_VEL
LIN {X 0,Y 58.021,Z 456.129,A -85,B 0,C 180,E1 -30614.266,E2 -30614.266} C_VEL
LIN {X 0,Y 51.458,Z 457.381,A -85,B 0,C 180,E1 -30617.02,E2 -30617.02} C_VEL
LIN {X 0,Y 38.838,Z 458.642,A -85,B 0,C 180,E1 -30625.171,E2 -30625.171} C_VEL
LIN {X 0,Y 27.819,Z 458.4,A -85,B 0,C 180,E1 -30640.686,E2 -30640.686} C_VEL
LIN {X 0,Y 23.633,Z 457.703,A -85,B 0,C 180,E1 -30653.468,E2 -30653.468} C_VEL
LIN {X 0,Y 21.002,Z 456.58,A -85,B 0,C 180,E1 -30670.414,E2 -30670.414} C_VEL
LIN {X 0,Y 20.31,Z 455.047,A -85,B 0,C 180,E1 -30689.963,E2 -30689.963} C_VEL
LIN {X 0,Y 21.981,Z 451.803,A -85,B 0,C 180,E1 -30718.617,E2 -30718.617} C_VEL
LIN {X 0,Y 27.628,Z 447.445,A -85,B 0,C 180,E1 -30739.693,E2 -30739.693} C_VEL
LIN {X 0,Y 35.665,Z 441.886,A -85,B 0,C 180,E1 -30752.41,E2 -30752.41} C_VEL
LIN {X 0,Y 44.716,Z 434.909,A -85,B 0,C 180,E1 -30760.497,E2 -30760.497} C_VEL
LIN {X 0,Y 52.759,Z 427.79,A -85,B 0,C 180,E1 -30764.888,E2 -30764.888} C_VEL
LIN {X 0,Y 61.017,Z 419.173,A -85,B 0,C 180,E1 -30768.16,E2 -30768.16} C_VEL
LIN {X 0,Y 66.872,Z 411.949,A -85,B 0,C 180,E1 -30770.059,E2 -30770.059} C_VEL
LIN {X 0,Y 74.54,Z 400.834,A -85,B 0,C 180,E1 -30771.777,E2 -30771.777} C_VEL
LIN {X 0,Y 80.53,Z 389.894,A -85,B 0,C 180,E1 -30772.956,E2 -30772.956} C_VEL
LIN {X 0,Y 85.736,Z 377.674,A -85,B 0,C 180,E1 -30773.852,E2 -30773.852} C_VEL
LIN {X 0,Y 89.656,Z 365.095,A -85,B 0,C 180,E1 -30774.443,E2 -30774.443} C_VEL
LIN {X 0,Y 92.173,Z 352.495,A -85,B 0,C 180,E1 -30774.869,E2 -30774.869} C_VEL
LIN {X 0,Y 93.489,Z 341.871,A -85,B 0,C 180,E1 -30775.213,E2 -30775.213} C_VEL
LIN {X 0,Y 92.965,Z 339.573,A -85,B 0,C 180,E1 -30778.376,E2 -30778.376} C_VEL
LIN {X 0,Y 92.686,Z 337.879,A -85,B 0,C 180,E1 -30781.289,E2 -30781.289} C_VEL
LIN {X 0,Y 92.541,Z 337.005,A -85,B 0,C 180,E1 -30784.356,E2 -30784.356} C_VEL
LIN {X 0,Y 92.653,Z 338.294,A -85,B 0,C 180,E1 -30790.547,E2 -30790.547} C_VEL
LIN {X 0,Y 93.35,Z 341.435,A -85,B 0,C 180,E1 -30795.848,E2 -30795.848} C_VEL
LIN {X 0,Y 93.445,Z 341.788,A -85,B 0,C 180,E1 -30796.327,E2 -30796.327} C_VEL
LIN {X 0,Y 91.101,Z 357.793,A -85,B 0,C 180,E1 -30796.848,E2 -30796.848} C_VEL
LIN {X 0,Y 87.965,Z 370.053,A -85,B 0,C 180,E1 -30797.48,E2 -30797.48} C_VEL
LIN {X 0,Y 83.265,Z 382.902,A -85,B 0,C 180,E1 -30798.547,E2 -30798.547} C_VEL
LIN {X 0,Y 77.532,Z 394.714,A -85,B 0,C 180,E1 -30799.917,E2 -30799.917} C_VEL
LIN {X 0,Y 70.865,Z 405.474,A -85,B 0,C 180,E1 -30801.645,E2 -30801.645} C_VEL
LIN {X 0,Y 63.327,Z 415.297,A -85,B 0,C 180,E1 -30803.755,E2 -30803.755} C_VEL
